Yaskawa INFORM job: OK_R2_O38-47,64(1)(90,180)OKKR.JBI

/JOB
//NAME OK_R2_O38-47,64(1)(90,180)OKKR
///FOLDERNAME X4
//POS
///NPOS 669,669,669,19,0,0
///TOOL 0
///POSTYPE PULSE
///PULSE
C00000=90909,-97924,-91406,33882,56334,-85304
C00001=105552,-103822,-93612,26444,49613,-80458
C00002=93803,-39674,-61862,-10952,72624,-83592
C00003=83044,29645,-6844,-3671,113202,-83073
C00004=80232,46018,13481,-1640,119259,-82796
C00005=84341,50404,17488,7249,115666,-79799
C00006=84629,52012,20689,7225,114506,-79766
C00007=84629,51890,21633,7182,113865,-79809
C00008=84629,52012,20689,7225,114506,-79766
C00009=84940,55701,25098,7229,113667,-79705
C00010=84940,55628,25812,7200,113194,-79735
C00011=84829,53963,24073,7195,113413,-79762
C00012=84779,55348,25092,7189,113502,-79775
C00013=83953,58737,25467,6224,116924,-79977
C00014=90636,-6579,-39383,-4621,91502,-82162
C00015=107016,-16132,-49825,-8384,94240,-77109
C00016=106659,-18282,-50653,15937,87636,-73637
C00017=135463,84611,26036,8427,98138,-63561
C00018=135459,73950,19227,14779,115232,-60625
C00019=121103,67404,21507,14676,120976,-65247
C00020=121102,66967,23101,14477,119807,-65411
C00021=121102,66637,23738,14388,119264,-65486
C00022=121102,66967,23101,14477,119807,-65411
C00023=120221,69773,26406,14234,119379,-65811
C00024=120221,69412,27152,14135,118755,-65896
C00025=120511,68181,25704,14224,118959,-65756
C00026=120221,69412,27152,14135,118755,-65896
C00027=120195,60975,7913,14673,121769,-65482
C00028=135454,84776,26243,8428,98096,-63567
C00029=106659,-18282,-50653,15937,87636,-73637
C00030=89310,-122172,-106686,13361,50676,-45199
C00031=123165,-113898,-119110,-19125,43336,19368
C00032=123668,-102412,-109547,-19577,43467,19587
C00033=131184,63359,57441,-15233,67840,18691
C00034=122068,78147,74274,-12505,69533,15106
C00035=122051,87849,89370,-12875,65325,15559
C00036=122051,89227,92048,-12969,64408,15664
C00037=122316,85057,86118,-12868,65923,15592
C00038=122667,82911,83414,-12880,66527,15655
C00039=122667,83831,85320,-12946,65844,15732
C00040=122426,86931,89254,-12983,65000,15737
C00041=122963,79390,78884,-12845,67528,15654
C00042=130632,64185,60223,-15235,66493,18662
C00043=131662,58983,54996,-15425,67212,18954
C00044=131668,55339,42428,-14901,72880,18222
C00045=146861,-92393,-105699,-36485,53490,27620
C00046=148000,-101656,-114811,-36865,54640,27702
C00047=148000,-101656,-114811,-36865,54640,27702
C00048=148000,-101656,-114811,-36865,54640,27702
C00049=159496,-161049,-136264,-30615,73499,21221
C00050=103228,-122632,-133352,7038,92284,523
C00051=103228,-122632,-133352,7038,92284,523
C00052=103228,-124480,-131601,7026,90271,411
C00053=103391,-121920,-131082,6996,91247,517
C00054=103853,-115329,-128981,6922,93290,780
C00055=103391,-120798,-132087,7006,92433,583
C00056=104641,-114737,-130152,6774,94243,1084
C00057=104641,-114737,-130152,6774,94243,1084
C00058=104641,-116137,-129119,6762,92896,1012
C00059=104641,-115940,-129279,6764,93095,1023
C00060=105111,-108950,-126961,6694,95208,1287
C00061=104576,-115792,-130426,6785,93876,1044
C00062=103741,-127928,-135528,6927,90867,609
C00063=103741,-127928,-135528,6927,90867,609
C00064=103741,-127928,-135528,6927,90867,609
C00065=103865,-116944,-129962,6921,93061,771
C00066=103865,-118485,-128547,6909,91408,679
C00067=103865,-118011,-129031,6913,91946,709
C00068=104350,-111197,-126797,6823,94018,978
C00069=103645,-119716,-131347,6963,92509,670
C00070=126331,-111187,-127566,2170,93341,7936
C00071=126314,-110675,-127191,2173,93374,7931
C00072=126314,-111741,-126360,2171,92316,7913
C00073=126314,-111248,-126762,2172,92816,7922
C00074=126152,-104604,-124481,2216,94828,7909
C00075=126314,-111061,-126906,2173,93001,7925
C00076=125902,-111149,-126935,2263,92984,7794
C00077=132196,-109284,-126305,-2386,93568,14490
C00078=132014,-110397,-125220,-2342,92324,14457
C00079=132014,-111538,-124094,-2340,91046,14481
C00080=132014,-110972,-124684,-2340,91699,14468
C00081=131346,-109003,-124013,-2196,92280,14246
C00082=132122,-112463,-125993,-2364,91740,14502
C00083=130696,-128652,-136015,-2037,89553,14081
C00084=130696,-128652,-136015,-2037,89553,14081
C00085=134573,-129962,-127961,-2886,84044,15460
C00086=135247,-123905,-124729,-3029,85191,15657
C00087=135247,-124242,-122895,-3032,83891,15687
C00088=135059,-121526,-122583,-2986,85086,15595
C00089=134621,-115318,-120572,-2888,87018,15405
C00090=135273,-124345,-124575,-3033,84868,15671
C00091=101634,-140552,-130463,4330,80438,4385
C00092=100831,-135445,-127742,4507,81431,4148
C00093=100831,-135220,-126147,4516,80567,4118
C00094=100831,-135304,-126661,4513,80840,4129
C00095=101541,-127818,-124438,4340,83274,4455
C00096=100689,-136992,-128168,4541,80909,4084
C00097=101700,-117063,-135109,4321,95328,4920
C00098=101700,-117063,-135109,4321,95328,4920
C00099=107464,-106510,-121453,3057,92107,6652
C00100=105693,-105772,-119256,3437,91202,6062
C00101=105693,-106748,-117862,3435,89847,6024
C00102=105693,-106325,-118509,3436,90460,6041
C00103=104724,-99451,-116018,3652,92493,5788
C00104=105563,-106984,-120499,3466,91350,6023
C00105=97637,-124436,-133710,5150,90918,3458
C00106=101700,-117063,-135109,4321,95328,4920
C00107=101700,-117063,-135109,4321,95328,4920
C00108=113885,-115939,-123860,1658,88568,8649
C00109=113885,-115976,-123799,1658,88510,8649
C00110=113885,-116503,-122835,1658,87648,8639
C00111=113928,-115223,-122529,1647,88114,8658
C00112=114061,-111130,-121156,1620,89368,8717
C00113=113613,-117192,-124203,1715,88138,8556
C00114=77135,-109099,-124316,9289,94737,-2930
C00115=77964,-100968,-118468,9143,95217,-2626
C00116=77964,-101677,-117713,9127,94398,-2685
C00117=77964,-101560,-117850,9129,94540,-2675
C00118=78928,-97543,-116360,8967,95572,-2290
C00119=77908,-100245,-119438,9173,96179,-2574
C00120=71973,-123086,-130703,10190,92110,-4818
C00121=61369,-106979,-129386,-18745,110548,43775
C00122=54050,-118433,-122678,-29834,105379,66043
C00123=54050,-118432,-122677,-29849,105379,66042
C00124=52380,-128849,-120518,-29019,98947,67079
C00125=52380,-128559,-118965,-28945,98241,67262
C00126=52380,-128751,-119946,-28990,98681,67146
C00127=50245,-132811,-121152,-28917,96763,66805
C00128=52380,-128751,-119946,-28990,98681,67146
C00129=49374,-119498,-117890,-29381,100712,65454
C00130=49135,-119946,-117683,-29342,100317,65463
C00131=49135,-119959,-116418,-29258,99629,65643
C00132=49135,-119963,-116925,-29289,99902,65571
C00133=47420,-122909,-117861,-29192,98489,65269
C00134=49767,-118756,-118042,-29437,101266,65461
C00135=58824,-127197,-127906,-29549,105900,67783
C00136=58824,-127197,-127906,-29549,105900,67783
C00137=55789,-138532,-125635,-28743,98511,68512
C00138=54845,-137144,-123724,-28738,97781,68329
C00139=54845,-136558,-122036,-28679,97131,68490
C00140=54845,-136878,-122937,-28709,97474,68406
C00141=52687,-141381,-124200,-28678,95380,68093
C00142=56052,-135036,-125386,-28893,100051,68223
C00143=56052,-135036,-125386,-28893,100051,68223
C00144=54923,-136926,-123517,-28734,97796,68355
C00145=54923,-136449,-122129,-28684,97260,68488
C00146=54923,-136715,-122887,-28711,97551,68416
C00147=52628,-141500,-124230,-28677,95326,68085
C00148=54923,-138669,-131970,-29176,101590,67387
C00149=49576,-128334,-132403,-27234,106270,69223
C00150=44922,-139442,-128392,-26353,97465,69516
C00151=43106,-142181,-127565,-26251,95168,69348
C00152=43106,-141292,-125343,-26201,94348,69532
C00153=43106,-141708,-126356,-26223,94717,69449
C00154=42222,-150085,-128620,-26118,91814,69764
C00155=43106,-141708,-126356,-26223,94717,69449
C00156=58006,-149727,-131155,-24086,101568,78058
C00157=67130,-160484,-130477,-19696,102779,86761
C00158=65530,-164092,-131264,-20694,100171,85228
C00159=25938,-108868,-115377,-27148,106727,70167
C00160=30236,-167786,-131335,-27861,77157,62843
C00161=40913,-181249,-136978,-30366,76641,63974
C00162=31337,-124593,-132531,-25311,107075,53461
C00163=107165,-96970,-126665,3187,100215,6761
C00164=107165,-106401,-121090,3121,91950,6553
C00165=98999,-123975,-120325,10477,76714,-326
C00166=104449,-120152,-119012,8815,77213,1590
C00167=136338,-77147,-102883,-1281,87901,12266
C00168=129257,-75496,-102169,6212,88982,4910
C00169=138081,-104464,-122106,-1833,85725,12838
C00170=119260,-105046,-123410,8534,87528,2432
C00171=124620,-151805,-134891,7305,72242,3267
C00172=124614,-151414,-134787,7302,72378,3273
C00173=124612,-151215,-134734,7300,72449,3276
C00174=124620,-151805,-134891,7305,72242,3267
C00175=127969,-108981,-129625,6073,90620,5362
C00176=128058,-112032,-130642,6044,89675,5344
C00177=99990,-117497,-120264,13536,83880,-4252
C00178=95862,-116029,-118012,14517,83962,-5647
C00179=139101,-101989,-113180,2891,83526,8647
C00180=134512,-124069,-125019,4259,79673,7022
C00181=124704,-125859,-130096,7035,82535,3892
C00182=99313,-127153,-133045,-12119,95446,32872
C00183=57886,-133831,-130402,-29291,103936,67934
C00184=55789,-138532,-125635,-28743,98511,68512
C00185=48693,-117877,-116324,-29063,104784,69163
C00186=50073,-120833,-117390,-28223,106210,71565
C00187=68626,-163926,-129258,-19114,104295,87122
C00188=70376,-133538,-127464,-20847,118406,85282
C00189=70376,-133538,-127464,-20847,118406,85282
C00190=56915,-96442,-108782,-30239,105442,63415
C00191=56121,-79134,-101591,-31100,116741,68778
C00192=90261,-137084,-122094,-21625,111979,84005
C00193=77475,-118139,-116359,-17026,122373,89952
C00194=79183,-112936,-123408,-17693,125433,82686
C00195=81561,-124200,-134149,-21063,125175,90603
C00196=103376,-109759,-132308,3968,97270,5504
C00197=101634,-140552,-130463,4330,80438,4385
C00198=110110,-127209,-124061,-3201,83105,15977
C00199=90594,-117032,-120596,11082,89723,-6771
C00200=125366,-116446,-120359,4331,86595,4547
C00201=114221,-95322,-113096,13979,98696,-11684
C00202=109678,-119625,-133746,14623,99658,-13079
C00203=112326,-124641,-135293,14185,97639,-12436
C00204=113675,-111285,-124420,14007,97585,-11993
C00205=113699,-111426,-124467,14002,97539,-11990
C00206=124004,-129907,-130136,8507,87303,-2218
C00207=139431,-131601,-130697,-461,84652,11785
C00208=149048,-100082,-120338,-2575,94643,14766
C00209=149098,-100150,-120363,-2585,94625,14781
C00210=144513,-99899,-120272,-1580,94586,13343
C00211=148184,-92878,-117624,-2396,96648,14454
C00212=154718,-145008,-134516,-3815,80522,16974
C00213=155631,-143491,-134098,-4008,81086,17267
C00214=123104,-120086,-121421,6334,85998,1376
C00215=127889,-117088,-120449,5327,86600,2988
C00216=148175,-95724,-112847,963,92122,9694
C00217=137316,-91860,-109869,13618,92576,-296
C00218=127829,-127486,-128792,15513,87749,-4031
C00219=127829,-122446,-134816,15592,93826,-3264
C00220=125285,-108995,-105645,-24533,66859,22374
C00221=121876,-100663,-100590,-22961,66967,21017
C00222=120611,-97454,-98556,-22372,66992,20522
C00223=120728,-95778,-96365,-22498,66572,20652
C00224=120611,-97454,-98556,-22372,66992,20522
C00225=120972,-98646,-98782,-22597,66650,20731
C00226=119814,-94892,-97816,-21908,67582,20099
C00227=120972,-98646,-98782,-22597,66650,20731
C00228=122255,-101873,-100811,-23195,66623,21236
C00229=125713,-110249,-105850,-24792,66512,22621
C00230=125414,-109454,-110952,-25434,70557,21724
C00231=121886,-100912,-105844,-23885,70668,20357
C00232=120575,-97642,-103795,-23303,70688,19860
C00233=120636,-96154,-101667,-23400,70203,19982
C00234=120575,-97642,-103795,-23303,70688,19860
C00235=121028,-97980,-103315,-23548,70382,20093
C00236=119871,-93906,-102218,-22897,71374,19458
C00237=121028,-97980,-103315,-23548,70382,20093
C00238=122351,-101230,-105354,-24132,70373,20595
C00239=125908,-109706,-110431,-25687,70298,21973
C00240=125468,-108852,-114009,-26132,73198,21211
C00241=121864,-100250,-108878,-24604,73277,19846
C00242=120523,-96969,-106822,-24029,73283,19350
C00243=120543,-95651,-104748,-24106,72739,19471
C00244=120523,-96969,-106822,-24029,73283,19350
C00245=121096,-97384,-106424,-24308,73024,19616
C00246=119937,-93066,-105230,-23683,74062,18974
C00247=121096,-97384,-106424,-24308,73024,19616
C00248=122450,-100644,-108468,-24886,73032,20117
C00249=126090,-109173,-113564,-26418,72994,21493
C00250=126107,-105383,-120588,-25792,78658,20214
C00251=115870,-101424,-121533,41206,90180,3452
C00252=115851,-106682,-115012,41260,85065,1433
C00253=119242,-98694,-109765,40357,84214,2540
C00254=120508,-95652,-107669,40003,83867,2939
C00255=120512,-93942,-105232,40036,83383,2757
C00256=120508,-95652,-107669,40003,83867,2939
C00257=119976,-95300,-106376,40178,83625,2624
C00258=123146,-93912,-105979,39274,82602,3565
C00259=119976,-95300,-106376,40178,83625,2624
C00260=118706,-98291,-108457,40527,83992,2228
C00261=115305,-106116,-113657,41413,84900,1133
C00262=117529,-113204,-110114,15038,59483,-16836
C00263=119860,-102582,-104476,13511,61010,-15725
C00264=120710,-98611,-102232,12973,61516,-15338
C00265=120712,-96036,-99318,13028,61058,-15391
C00266=120710,-98611,-102232,12973,61516,-15338
C00267=120133,-97446,-101425,13271,61707,-15536
C00268=121539,-92419,-99938,12330,63118,-14842
C00269=120133,-97446,-101425,13271,61707,-15536
C00270=119274,-101350,-103659,13810,61233,-15923
C00271=116924,-111770,-109266,15331,59803,-17031
C00272=118012,-90030,-113480,10859,76824,-11039
C00273=121151,-43618,-104634,-1145,105190,4571
C00274=120753,-40362,-99446,-1000,103667,4481
C00275=120604,-39041,-97355,-946,103057,4446
C00276=120606,-40163,-95662,-941,101440,4458
C00277=120604,-39041,-97355,-946,103057,4446
C00278=120772,-35445,-95769,-1008,103931,4483
C00279=120462,-29091,-92658,-908,105279,4391
C00280=120772,-35445,-95769,-1008,103931,4483
C00281=120921,-36668,-97839,-1062,104577,4517
C00282=121319,-39651,-102962,-1210,106200,4605
C00283=108629,-121399,-122702,16889,67135,-14241
C00284=115336,-113367,-105488,19088,53546,-18271
C00285=117865,-102996,-100223,17109,54980,-16930
C00286=118786,-99066,-98108,16412,55481,-16461
C00287=118815,-96798,-95161,16518,54853,-16552
C00288=118786,-99066,-98108,16412,55481,-16461
C00289=119112,-97264,-98148,16039,56331,-16193
C00290=118757,-93015,-97035,15990,57843,-16106
C00291=119112,-97264,-98148,16039,56331,-16193
C00292=123316,-98367,-98161,13561,55035,-14648
C00293=126858,-97217,-97820,11275,54872,-13210
C00294=123316,-98367,-98161,13561,55035,-14648
C00295=122519,-102389,-100318,14180,54451,-15058
C00296=120328,-113051,-105701,15959,52759,-16243
C00297=124093,-110707,-95637,-16539,52225,18162
C00298=121727,-101468,-90458,-14864,53273,16967
C00299=120864,-97923,-88367,-14268,53637,16545
C00300=120864,-95769,-85768,-14357,53158,16613
C00301=120864,-97923,-88367,-14268,53637,16545
C00302=120753,-94948,-87925,-13988,54838,16331
C00303=119636,-91806,-87160,-13170,55764,15745
C00304=120753,-94948,-87925,-13988,54838,16331
C00305=121593,-98445,-90034,-14553,54501,16732
C00306=123889,-107558,-95262,-16133,53518,17861
C00307=123907,-109460,-104253,-15319,57915,17198
C00308=120718,-89127,-94408,93,103364,-81793
C00309=120702,-88967,-86044,90,98299,-81802
C00310=120714,-92346,-83648,90,95088,-81800
C00311=120719,-93530,-82604,90,93837,-81800
C00312=120721,-91291,-79709,90,93204,-81799
C00313=120719,-93530,-82604,90,93837,-81800
C00314=120503,-94372,-82680,81,93451,-81873
C00315=120503,-97134,-83277,81,92401,-81874
C00316=120503,-94372,-82680,81,93451,-81873
C00317=120501,-93212,-83739,81,94699,-81873
C00318=120496,-89894,-86173,82,97902,-81873
C00319=120512,-90208,-94601,84,102927,-81864
C00320=120739,-87258,-85833,92,99047,-81789
C00321=120752,-90752,-83510,91,95822,-81787
C00322=120758,-91982,-82493,91,94564,-81786
C00323=120759,-89478,-79257,91,93861,-81786
C00324=120758,-91982,-82493,91,94564,-81786
C00325=120462,-95334,-83503,80,93464,-81887
C00326=120461,-97919,-84058,79,92477,-81888
C00327=120462,-95334,-83503,80,93464,-81887
C00328=120460,-94163,-84562,80,94717,-81887
C00329=120456,-90813,-86994,80,97935,-81887
C00330=121033,-93279,-128320,-140,99068,4698
C00331=120997,-110061,-117241,-128,83627,4703
C00332=120579,-101211,-110995,-15,84330,4566
C00333=120424,-97983,-108548,25,84483,4515
C00334=120430,-96385,-106046,24,83763,4517
C00335=120424,-97983,-108548,25,84483,4515
C00336=120936,-92390,-106244,-111,85940,4681
C00337=120538,-86818,-104536,-4,87751,4552
C00338=120936,-92390,-106244,-111,85940,4681
C00339=121096,-95373,-108656,-154,85891,4732
C00340=121527,-103462,-114785,-270,85508,4872
C00341=75677,-91018,-121004,38809,104477,3256
C00342=86494,-89564,-122641,29897,102391,4704
C00343=121241,-108971,-117698,-1136,79653,4828
C00344=120728,-99263,-111358,-963,80734,4651
C00345=120539,-95742,-108880,-900,81016,4587
C00346=120543,-94296,-106552,-902,80326,4593
C00347=120539,-95742,-108880,-900,81016,4587
C00348=120728,-93992,-107595,-961,81127,4647
C00349=120728,-90301,-106424,-959,82303,4638
C00350=120728,-93992,-107595,-961,81127,4647
C00351=121024,-97533,-112143,-1058,82109,4735
C00352=121551,-107098,-118478,-1235,81100,4915
C00353=121569,-100080,-124444,-1231,88376,4850
C00354=117898,-83225,-110918,12916,113641,-67504
C00355=119870,-90654,-110250,12481,109228,-67312
C00356=120686,-93336,-109842,12338,107519,-67211
C00357=120688,-92183,-107571,12276,106730,-67294
C00358=120686,-93336,-109842,12338,107519,-67211
C00359=120163,-91649,-109473,12395,108219,-67318
C00360=121681,-97188,-111137,12239,106219,-67001
C00361=120163,-91649,-109473,12395,108219,-67318
C00362=119359,-88923,-109851,12543,109932,-67413
C00363=117416,-81399,-110449,12994,114344,-67589
C00364=120617,-94125,-108136,-8857,121741,-88541
C00365=120616,-94449,-107526,-8800,121205,-88496
C00366=136098,-107181,-107429,-16269,112846,-84409
C00367=120444,-95183,-107742,-8816,120947,-88541
C00368=119761,-91680,-105499,-9024,121288,74873
C00369=120616,-95784,-105179,19399,105655,-65758
C00370=120617,-94769,-108163,19676,107886,-65380
C00371=121686,-93853,-106574,24019,104588,-57765
C00372=120617,-92780,-110041,24421,107344,-57569
C00373=120617,-90665,-112384,24828,109654,-57058
C00374=120619,-82046,-117525,26421,116533,-55408
C00375=120645,-81988,-112872,3577,88664,-15070
C00376=120614,-96077,-90479,-12976,48732,14983
C00377=120612,-93911,-81283,-13967,44304,15634
C00378=120612,-93390,-79613,-14157,43566,15753
C00379=121252,-93346,-79166,-14714,43437,16096
C00380=121500,-95247,-79374,-15137,42660,16355
C00381=120782,-94947,-80724,-14317,43483,15851
C00382=120611,-93982,-79716,-14233,43318,15795
C00383=120612,-95725,-83890,-13821,44941,15536
C00384=121326,-94847,-83951,-14224,45559,15784
C00385=120613,-94980,-84633,-13612,45776,15407
C00386=120613,-95388,-86250,-13438,46540,15293
C00387=120616,-96933,-104006,5046,49827,739
C00388=120616,-97132,-103061,5097,49146,704
C00389=120617,-95323,-101728,5088,49256,711
C00390=120871,-100699,-104338,4972,48087,759
C00391=120795,-98262,-101888,5054,47837,712
C00392=120618,-95198,-103493,5003,50401,770
C00393=121122,-95129,-103646,4600,50501,986
C00394=120617,-97030,-104927,5009,50342,766
C00395=120617,-96757,-105844,4959,51045,801
C00396=120618,-92718,-112658,4589,57292,1090
C00397=108098,-105677,-132023,7461,89264,-328
C00398=80455,-75739,-120669,16714,100968,-7375
C00399=97258,-84752,-105297,10869,90674,-3530
C00400=97358,-86422,-102930,10833,88387,-3696
C00401=97424,-86715,-102018,10818,87679,-3736
C00402=97216,-90521,-102980,10875,86365,-3919
C00403=97404,-84940,-102216,10822,88698,-3655
C00404=120617,-94266,-106774,4665,84598,3614
C00405=111454,-84543,-103018,13521,90962,-7073
C00406=109783,-86139,-104921,12729,90791,-5985
C00407=106092,-100123,-116923,13597,91547,-7106
C00408=102052,-116072,-128299,14497,91044,-8487
C00409=91007,-121504,-125767,15485,91359,-21712
C00410=120613,-95050,-86060,3557,95049,-80550
C00411=120612,-93945,-81838,3544,93023,-80607
C00412=121155,-91942,-79314,3616,92478,-80448
C00413=120652,-94806,-81837,3543,92579,-80606
C00414=120610,-90975,-79567,3544,93151,-80605
C00415=150255,-82598,-75582,4413,93505,-70504
C00416=122384,-91795,-77981,11848,92227,-69969
C00417=120612,-93489,-79991,12120,92904,-70125
C00418=120613,-94640,-84016,12161,94749,-69944
C00419=120614,-96377,-93023,12320,99298,-69491
C00420=120644,-125570,-121052,-6784,67869,-5403
C00421=120615,-96622,-98748,-12572,58745,14095
C00422=120615,-96643,-96984,-12717,57674,14222
C00423=127606,-89142,-93330,-20657,62312,19456
C00424=120926,-99715,-97034,-13118,56212,14526
C00425=120613,-97817,-97899,-12721,57634,14225
C00426=120615,-96818,-95655,6616,54391,866
C00427=120615,-97044,-96976,6561,55085,910
C00428=112093,-90513,-93108,22044,58833,-17349
C00429=120615,-96644,-96112,9528,53512,-9485
C00430=120615,-96653,-97679,9416,54459,-9397
C00431=120616,-95373,-105489,8868,59856,-8934
C00432=117333,-91440,-108817,14098,83709,-30265
C00433=112347,-94381,-87846,22750,99580,-64599
C00434=112329,-92021,-78548,22454,95406,-65402
C00435=115628,-91274,-75119,22621,92902,-64661
C00436=117255,-90241,-73175,22718,91835,-64269
C00437=117028,-88603,-73220,22719,92705,-64185
C00438=116923,-92272,-75451,22697,92259,-64308
C00439=120553,-90828,-77383,-15099,94128,-70510
C00440=120613,-90885,-77384,-15804,94030,-70628
C00441=123770,-105111,-82751,-16580,84167,-79857
C00442=124886,-104010,-85216,-16560,86394,-79763
C00443=120613,-94284,-84162,-15892,96365,-70931
C00444=120614,-95920,-93129,-16139,100869,-71526
C00445=120649,-92160,-111225,-3199,84919,-49711
C00446=120616,-97604,-99172,11891,40402,-23254
C00447=120614,-96911,-90603,13253,35598,-24030
C00448=120614,-96763,-89737,13401,35153,-24111
C00449=121291,-96342,-89250,12683,34963,-23744
C00450=119113,-97762,-90324,15090,35268,-24978
C00451=120705,-99580,-90146,13704,33974,-24279
C00452=121588,-95238,-86691,12692,33949,-23762
C00453=127502,-77730,-88040,-1756,56127,-19882
C00454=125086,-93679,-98074,-150,54079,-20822
C00455=120613,-95818,-85653,14108,33181,-24494
C00456=120615,-97479,-97669,6545,55280,923
C00457=121580,-96410,-96097,5967,54791,1285
C00458=120928,-100587,-97757,6468,53722,953
C00459=120613,-98670,-98620,6548,55254,920
C00460=120615,-96854,-96360,6584,54805,893
C00461=120615,-97074,-97513,6537,55399,931
C00462=114077,-92170,-94328,19163,57465,-15491
C00463=120615,-97626,-97578,9481,53904,-9448
C00464=120636,-112691,-117418,8831,59265,-10492
C00465=120617,-94408,-109491,7961,65698,-13071
C00466=120616,-97035,-102174,8375,59902,-13490
C00467=120616,-97254,-100452,8474,58742,-13580
C00468=120616,-96110,-99125,8495,58514,-13598
C00469=120614,-98453,-101360,8481,58685,-13585
C00470=119727,-100186,-100479,9138,57364,-14041
C00471=120617,-96158,-99373,8483,58642,-13587
C00472=120616,-97215,-100721,8458,58926,-13566
C00473=120616,-96978,-102436,8360,60091,-13476
C00474=120617,-94247,-109716,7948,65917,-13056
C00475=120616,-96445,-103082,-5252,59171,13430
C00476=120615,-96888,-94956,-5569,53965,13694
C00477=120614,-96711,-93127,-5642,52935,13750
C00478=120614,-96618,-92386,-5672,52529,13773
C00479=119756,-94067,-91753,-5051,53390,13370
C00480=120525,-97964,-94062,-5589,52861,13717
C00481=120614,-96681,-92800,-5656,52750,13760
C00482=120614,-96709,-92988,-5648,52851,13755
C00483=120614,-96767,-93400,-5632,53074,13742
C00484=120614,-96843,-94134,-5603,53484,13720
C00485=120615,-96977,-95945,-5531,54526,13664
C00486=120616,-97003,-101109,-6851,58481,13557
C00487=120615,-97139,-99377,-6934,57353,13629
C00488=120615,-97164,-98672,-6968,56909,13657
C00489=119756,-94335,-97933,-6375,57832,13263
C00490=120570,-98373,-100300,-6912,57283,13615
C00491=120615,-97165,-99156,-6946,57204,13638
C00492=120616,-97129,-99856,-6912,57651,13610
C00493=120616,-96964,-101578,-6829,58787,13537
C00494=120617,-96349,-105255,-7716,61917,13386
C00495=120616,-96771,-103611,-7804,60699,13471
C00496=120616,-96905,-102940,-7840,60222,13505
C00497=119756,-93851,-102113,-7266,61195,13116
C00498=120602,-97980,-104523,-7800,60639,13470
C00499=120616,-96844,-103353,-7819,60505,13485
C00500=120616,-96699,-104019,-7783,60985,13451
C00501=120617,-96245,-105652,-7696,62212,13366
C00502=120618,-92150,-112439,-7334,68442,12961
C00503=130920,-122289,-127601,23263,76296,-33617
C00504=126647,-121486,-124764,14921,71090,-19914
C00505=118673,-117816,-113052,9081,54805,-1270
C00506=119719,-97166,-102733,8035,58912,-525
C00507=118944,-92090,-109805,27006,83902,-36269
C00508=120616,-93914,-111601,26462,83549,-35758
C00509=120617,-94475,-108119,24525,75199,-30020
C00510=120618,-90011,-113520,23738,94905,-43572
C00511=120617,-93534,-109718,22404,79768,-31867
C00512=120617,-93028,-110386,24696,84592,-28860
C00513=120617,-93859,-109223,24523,82429,-27907
C00514=120617,-95217,-106728,22357,73913,-21133
C00515=120616,-96198,-104144,16550,64688,-11231
C00516=120616,-97587,-102867,7505,58697,-196
C00517=120615,-98378,-102979,-677,57412,8649
C00518=120615,-98092,-104435,-2505,58558,10610
C00519=120615,-97859,-104607,-2041,58746,10113
C00520=120615,-97689,-104685,-1580,58853,9618
C00521=120615,-97267,-104663,2078,59079,5700
C00522=122185,-96113,-104438,1107,59504,6297
C00523=124417,-94235,-103728,-259,60020,7133
C00524=120617,-96195,-105273,2057,60007,5718
C00525=120617,-95777,-106468,2039,60956,5736
C00526=120690,-30346,-78642,-22937,64170,21118
C00527=120690,-30346,-78642,-22937,64170,21118
C00528=98469,-5770,-79404,-6171,73775,13621
C00529=73961,-64832,-115099,11040,66386,6438
C00530=152983,-151482,-105999,-63266,53723,-19798
C00531=133395,-32083,-56059,-41211,61963,-37621
C00532=138234,23065,45169,-67508,45202,-44915
C00533=136781,30072,55747,-70235,43147,-43411
C00534=136213,33214,60449,-71542,42329,-42699
C00535=136213,31591,57334,-70422,42710,-43384
C00536=136788,30891,57778,-71075,42855,-42892
C00537=134893,29619,56778,-71118,41623,-43172
C00538=133284,25640,52793,-70642,40733,-43707
C00539=131869,22445,49655,-70246,39929,-44150
C00540=132436,19576,45433,-69035,40713,-44782
C00541=133889,13007,35719,-66469,42691,-46136
C00542=120930,8852,32410,-71146,24358,-44597
C00543=120056,16713,42856,-76185,23038,-42237
C00544=121640,23151,50001,-78915,23835,-40720
C00545=120179,17981,45384,-78314,22894,-41190
C00546=119718,18730,44666,-76295,22791,-42223
C00547=126194,31546,58401,-80948,26724,-39140
C00548=125034,24898,50699,-78244,26224,-40637
C00549=126001,16678,39521,-73266,27604,-43020
C00550=110893,28996,24386,-6920,61269,-70362
C00551=121937,-147756,-98721,-13314,47766,-64479
C00552=71720,-152863,-104081,12596,70757,-83485
C00553=71720,-152863,-104081,12596,70757,-83485
C00554=91982,-28216,-51992,-2303,92813,-79298
C00555=103376,51680,-13547,-11468,103274,-76678
C00556=78528,58148,26133,-1884,110066,-82404
C00557=73446,48868,27968,6188,106692,-82975
C00558=73676,48050,29892,6162,105078,-82976
C00559=73848,53549,43602,3176,111557,-82441
C00560=73910,56793,48494,3163,110214,-82456
C00561=74442,47740,29556,6278,105066,-82704
C00562=74442,47438,26373,6344,106859,-82610
C00563=75619,47557,26500,6517,106749,-82195
C00564=75166,47792,29439,6389,105108,-82446
C00565=75942,47613,29246,6502,105072,-82172
C00566=75379,35078,11730,9910,104528,-82166
C00567=80787,8835,-12135,-75,87858,-197
C00568=78204,48375,24964,11405,32429,78205
C00569=74266,-35048,-47468,15580,34736,76255
C00570=76186,-37462,-43585,14686,30875,76605
C00571=72421,-24340,-29465,20568,29825,73730
C00572=72122,-21014,-25782,21301,29384,73365
C00573=70865,-21091,-26712,22563,30208,72759
C00574=70738,-23036,-26859,23341,29404,72363
C00575=73032,-21271,-25966,20119,29138,73940
C00576=72310,-21659,-27383,20648,29949,73692
C00577=73400,-22218,-27785,19257,29646,74366
C00578=78913,-22240,-26725,-522,27359,85032
C00579=79845,-22599,-26982,-1923,27347,85705
C00580=74626,-21952,-29259,17095,30372,75430
C00581=71216,-28758,-34962,21414,31172,73342
C00582=77326,-37520,-49068,12046,33946,77926
C00583=83330,-46575,-52890,13958,55049,41505
C00584=86193,-52033,-54165,20785,79907,-1804
C00585=87571,-35325,-52921,25788,81678,-348
C00586=87508,-34952,-39783,27132,74543,-196
C00587=104644,32154,27534,-4448,60513,-72731
C00588=93805,201,18674,-23355,11914,-69008
C00589=93808,216,18686,-23365,11915,-69004
C00590=93810,222,18691,-23369,11915,-69002
C00591=93638,2355,20486,-22861,11860,-69245
C00592=93955,-2017,16089,-22978,12371,-69170
C00593=93808,210,18682,-23363,11914,-69005
C00594=93806,198,18671,-23357,11914,-69008
C00595=93804,186,18662,-23351,11913,-69011
C00596=93802,180,18657,-23347,11913,-69012
C00597=93799,166,18644,-23338,11912,-69017
C00598=93810,232,18700,-23265,11906,-69051
C00599=95314,-4751,13530,-26418,12915,-67513
C00600=95472,472,19818,-29385,11915,-66147
C00601=93990,-1863,16961,-23823,11950,-68785
C00602=93814,-607,16661,-21825,12670,-69707
C00603=101206,3306,22214,-43193,14297,-59419
C00604=100936,-4761,10472,-35572,16592,-62958
C00605=101724,-18723,-6868,-31140,19848,-65000
C00606=104644,32154,27534,-4448,60513,-72731
C00607=81813,-56841,-53371,53266,50302,-14082
C00608=60380,-131230,-84967,114894,34586,-40161
C00609=75788,-111312,-115723,41491,75595,-63087
C00610=90161,-54224,-109841,-7916,106787,-80704
C00611=104839,2947,-47825,-15873,91805,-74161
C00612=89900,18802,-35938,-9766,95357,-80687
C00613=83481,65005,13429,9056,119285,-78997
C00614=84379,59258,13120,8878,116463,-78905
C00615=105122,63991,30490,-2309,126100,-76457
C00616=105343,61862,26796,-2259,127285,-76391
C00617=86425,59542,13444,9048,116200,-78190
C00618=84859,64061,16437,8959,116837,-78702
C00619=84733,23156,-31643,6898,102580,-79911
C00620=89806,-37631,-52942,-13196,44828,-72538
C00621=94750,-32934,-45091,-18174,44929,-69862
C00622=95076,-26053,-35452,-19245,42727,-69219
C00623=107305,-33153,-35053,-31246,31625,-63156
C00624=107702,-34958,-34985,-32523,30946,-62498
C00625=98239,-24688,-34495,-21885,43616,-67814
C00626=95242,-30076,-40811,-18964,43932,-69406
C00627=95187,-81119,-79791,-20309,40550,-69551
C00628=116770,-29253,-58359,-25644,67366,-65351
C00629=114505,57687,20883,1024,117266,-70683
C00630=114650,58283,25572,1570,115664,-70627
C00631=114340,74668,47492,6514,119432,-70541
C00632=114056,77377,51999,6323,118081,-70732
C00633=114904,58629,25963,1620,115597,-70533
C00634=114904,58844,24763,1634,116445,-70521
C00635=115700,60684,26853,1789,116088,-70230
C00636=115527,59563,26959,1744,115454,-70303
C00637=116183,60608,28143,1870,115246,-70063
C00638=116183,61347,24564,1918,117826,-70018
C00639=115340,32559,-12600,852,114283,-70930
C00640=136323,52272,9545,-44589,64919,-61463
C00641=135074,-39507,-20212,-67575,45484,-47636
C00642=135318,-36807,-17542,-67853,45540,-47442
C00643=132787,-33499,-8836,-71025,42480,-45664
C00644=136770,-25555,-2359,-71345,45178,-45070
C00645=137559,-27867,-5282,-70853,45921,-45309
C00646=137893,-26315,-4086,-70829,46171,-45290
C00647=138309,-31340,-10754,-69522,47005,-46113
C00648=134147,-41542,-18435,-69427,44030,-46529
C00649=141128,-29133,-31085,-43489,44991,-50173
C00650=141423,-23417,-25276,-46918,44761,-56943
C00651=142721,-20298,-19655,-49027,44184,-55636
C00652=146072,-18893,-14822,-60688,47208,-48761
C00653=145286,-17068,-12207,-60970,46372,-48581
C00654=147042,-10361,-12167,-50830,46887,-54547
C00655=146980,-8744,-14162,-48811,51872,-51880
C00656=141391,-26070,-33699,-44316,51156,-54843
C00657=135350,-43982,-50251,-40364,49000,-57185
C00658=135985,2271,-36804,9338,77862,-64370
C00659=125855,24131,-11164,15237,94532,-65211
C00660=127405,33399,-2104,16711,101562,-63562
C00661=127405,32756,72,16600,99959,-63785
C00662=132541,67844,41901,19973,110951,-60327
C00663=132116,69898,43068,19947,111372,-60417
C00664=131318,40837,8366,16232,98288,-62662
C00665=131725,32981,-1351,15245,94948,-63065
C00666=135145,-3466,-36539,10688,79487,-64114
C00667=125690,-78122,-87562,13631,67908,-68588
C00668=2173,-78122,-87562,13631,67908,-68588
BC00000=277574,497829,168108
BC00001=277574,439333,87994
BC00002=272426,396216,154258
BC00003=276020,397785,163842
BC00004=276959,398195,166346
BC00005=274741,403082,149056
BC00006=274741,403082,149056
BC00007=274741,403082,149056
BC00008=274741,403082,149056
BC00009=274741,403082,149056
BC00010=274741,403082,149056
BC00011=274741,403082,149056
BC00012=274741,403082,149056
BC00013=275374,402065,146063
BC00014=277200,399025,164359
BC00015=277200,399025,164359
BC00016=277574,398402,168108
BC00017=337058,429692,17
BC00018=337058,399419,13781
BC00019=288570,380415,46933
BC00020=288570,380415,46933
BC00021=288570,380415,46933
BC00022=288570,380415,46933
BC00023=288570,380415,46933
BC00024=288570,380415,46933
BC00025=288570,380415,46933
BC00026=288570,380415,46933
BC00027=288570,380415,46933
BC00028=326292,423556,17
BC00029=277574,398402,168108
BC00030=248570,470524,121847
BC00031=96843,506307,308542
BC00032=96843,434340,293706
BC00033=128699,374993,308542
BC00034=128699,360593,308542
BC00035=128699,360593,308542
BC00036=128699,360593,308542
BC00037=128699,360593,308542
BC00038=128699,360593,308542
BC00039=128699,360593,308542
BC00040=128699,360593,308542
BC00041=128699,360593,308542
BC00042=128699,370385,308542
BC00043=128699,370385,308542
BC00044=128699,370385,308542
BC00045=128699,434340,293706
BC00046=128699,506307,308542
BC00047=128699,506307,1074774
BC00048=128699,506307,1074774
BC00049=10685,307107,1074774
BC00050=2446,176929,1073423
BC00051=90,176033,1058429
BC00052=90,176033,1058429
BC00053=90,176033,1058429
BC00054=90,176033,1058429
BC00055=90,176033,1058429
BC00056=75724,192083,1061957
BC00057=76484,191603,1056714
BC00058=76484,191603,1056714
BC00059=76484,191603,1056714
BC00060=76484,191603,1056714
BC00061=76484,191603,1056714
BC00062=76484,191603,1056714
BC00063=62310,231239,1056714
BC00064=67554,227591,1021238
BC00065=67554,227591,1021238
BC00066=67554,227591,1021238
BC00067=67554,227591,1021238
BC00068=67554,227591,1021235
BC00069=67554,227591,1021238
BC00070=67554,227591,1021238
BC00071=67554,227591,1021238
BC00072=67554,227591,1021238
BC00073=67554,227591,1021238
BC00074=67554,227591,1021238
BC00075=67554,227591,1021238
BC00076=145464,246213,1073324
BC00077=166805,220817,1072040
BC00078=166805,220817,1072040
BC00079=166805,220817,1072040
BC00080=166805,220817,1072040
BC00081=166805,220817,1072040
BC00082=166805,220817,1072040
BC00083=166804,220816,1072039
BC00084=274112,228208,1072039
BC00085=274112,228208,1072039
BC00086=274112,228208,1072039
BC00087=274112,228208,1072039
BC00088=274112,228208,1072039
BC00089=274112,228208,1072039
BC00090=274112,228208,1072039
BC00091=274112,228208,1072039
BC00092=274112,228208,1072035
BC00093=274112,228208,1072035
BC00094=274112,228208,1072035
BC00095=274112,228208,1072035
BC00096=274112,228208,1072035
BC00097=274112,228208,1072035
BC00098=253771,294542,1072035
BC00099=253771,294542,1066351
BC00100=253771,294542,1066351
BC00101=253771,294542,1066351
BC00102=253771,294542,1066351
BC00103=253771,294542,1066351
BC00104=253771,294542,1066351
BC00105=253771,294542,1066351
BC00106=332674,307450,1072035
BC00107=352760,246268,1062013
BC00108=352760,246268,1056084
BC00109=352760,246268,1056084
BC00110=352760,246268,1056084
BC00111=352760,246268,1056084
BC00112=352760,246268,1056084
BC00113=352760,246268,1056084
BC00114=352760,246268,1056084
BC00115=352760,246268,1056084
BC00116=352760,246268,1056084
BC00117=352760,246268,1056084
BC00118=352760,246268,1056084
BC00119=352760,246268,1056084
BC00120=352760,246268,1056084
BC00121=310153,278141,1073433
BC00122=291607,278327,1074936
BC00123=268886,285111,1073169
BC00124=268886,285111,1073169
BC00125=268886,285111,1073169
BC00126=268886,285111,1073169
BC00127=268886,285111,1073169
BC00128=268886,285111,1073169
BC00129=320862,285111,1073169
BC00130=320862,285111,1073169
BC00131=320862,285111,1073169
BC00132=320862,285111,1073169
BC00133=320862,285111,1073169
BC00134=320862,285111,1073169
BC00135=320862,285111,1073169
BC00136=213321,285111,1073169
BC00137=213321,285111,1068759
BC00138=213321,285111,1068759
BC00139=213321,285111,1068759
BC00140=213321,285111,1068759
BC00141=213321,285111,1068759
BC00142=213321,285111,1068759
BC00143=170741,285111,1068759
BC00144=170741,285111,1068759
BC00145=170741,285111,1068759
BC00146=170741,285111,1068759
BC00147=170741,285111,1068759
BC00148=170741,285111,1068759
BC00149=193205,122603,1068759
BC00150=193205,122603,1068759
BC00151=193205,122603,1068759
BC00152=193205,122603,1068759
BC00153=193205,122603,1068759
BC00154=193205,122603,1068759
BC00155=193205,122603,1068759
BC00156=199695,122603,1068758
BC00157=207772,122603,1068756
BC00158=207772,122603,1068754
BC00159=207772,122603,1068756
BC00160=207772,122603,1068756
BC00161=207772,122603,1068756
BC00162=207772,122603,1073551
BC00163=282390,309614,1068519
BC00164=282390,309614,1066351
BC00165=282388,309615,1066351
BC00166=282388,309615,1066351
BC00167=282388,309615,1066351
BC00168=282388,309615,1066351
BC00169=282388,309615,1066351
BC00170=100662,216693,1072303
BC00171=113337,188658,1072303
BC00172=107541,187687,1072404
BC00173=36523,175786,1073647
BC00174=30619,174782,1073647
BC00175=112223,231348,1072404
BC00176=388754,325280,1072404
BC00177=395558,265794,1072402
BC00178=396585,256820,1072402
BC00179=396585,256820,1072402
BC00180=396585,256820,1072402
BC00181=396585,256820,1072402
BC00182=316583,269170,1070812
BC00183=213321,285111,1068759
BC00184=213321,285111,1068759
BC00185=213321,285111,1068759
BC00186=213321,285111,1068759
BC00187=213321,285111,1068759
BC00188=213321,285111,1068759
BC00189=327369,285111,1068759
BC00190=316865,305805,1068759
BC00191=316865,305805,1068759
BC00192=316865,305805,1068759
BC00193=316865,305805,1068759
BC00194=316858,305779,1068759
BC00195=316082,302674,1068759
BC00196=274112,236301,1072039
BC00197=274112,228208,1072039
BC00198=274113,228208,1072037
BC00199=274113,228208,1072037
BC00200=274113,228208,1072037
BC00201=274113,228208,1072037
BC00202=274113,228208,1072037
BC00203=191168,215841,1072037
BC00204=191168,215841,1072037
BC00205=191168,215841,1072037
BC00206=191168,215841,1072037
BC00207=191168,215841,1072037
BC00208=191168,215841,1072037
BC00209=191168,215841,1072037
BC00210=181197,215841,1072037
BC00211=181197,215841,1072037
BC00212=181197,215841,1072037
BC00213=102071,227043,1072037
BC00214=102071,227043,1072037
BC00215=102071,227043,1072037
BC00216=102071,227043,1072037
BC00217=102071,227043,1072037
BC00218=102071,227043,1072034
BC00219=124217,449505,1070714
BC00220=168838,345562,1075139
BC00221=168838,345562,1075139
BC00222=168838,345562,1075139
BC00223=168838,345562,1075139
BC00224=168838,345562,1075139
BC00225=168838,345562,1075139
BC00226=168838,345562,1075139
BC00227=168838,345562,1075139
BC00228=168838,345562,1075139
BC00229=168838,345562,1075139
BC00230=125540,323298,1075139
BC00231=125540,323298,1075139
BC00232=125540,323298,1075139
BC00233=125540,323298,1075139
BC00234=125540,323298,1075139
BC00235=125540,323298,1075139
BC00236=125540,323298,1075139
BC00237=125540,323298,1075139
BC00238=125540,323298,1075139
BC00239=125540,323298,1075139
BC00240=94014,306720,1075139
BC00241=94014,306720,1075139
BC00242=94014,306720,1075139
BC00243=94014,306720,1075139
BC00244=94014,306720,1075139
BC00245=94014,306720,1075139
BC00246=94014,306720,1075139
BC00247=94014,306720,1075139
BC00248=94014,306720,1075139
BC00249=94014,306720,1075139
BC00250=94014,306720,1075139
BC00251=254000,289563,1075139
BC00252=254000,289563,1075139
BC00253=254000,289563,1075139
BC00254=254000,289563,1075139
BC00255=254000,289563,1075139
BC00256=254000,289563,1075139
BC00257=254000,289563,1075139
BC00258=254000,289563,1075139
BC00259=254000,289563,1075139
BC00260=254000,289563,1075139
BC00261=254000,289563,1075139
BC00262=131735,327892,1075139
BC00263=131735,327892,1075139
BC00264=131735,327892,1075139
BC00265=131735,327892,1075139
BC00266=131735,327892,1075139
BC00267=131735,327892,1075139
BC00268=131735,327892,1075139
BC00269=131735,327892,1075139
BC00270=131735,327892,1075139
BC00271=131735,327892,1075139
BC00272=107464,322487,1075139
BC00273=36166,306609,1075139
BC00274=36166,306609,1075139
BC00275=36166,306609,1075139
BC00276=36166,306609,1075139
BC00277=36166,306609,1075139
BC00278=36166,306609,1075139
BC00279=36166,306609,1075139
BC00280=36166,306609,1075139
BC00281=36166,306609,1075139
BC00282=36166,306609,1075139
BC00283=65350,327285,1075139
BC00284=79942,337624,1075139
BC00285=79942,337624,1075139
BC00286=79942,337624,1075139
BC00287=79942,337624,1075139
BC00288=79942,337624,1075139
BC00289=79942,337624,1075139
BC00290=79942,337624,1075139
BC00291=79942,337624,1075139
BC00292=79942,337624,1075139
BC00293=79942,337624,1075139
BC00294=79942,337624,1075139
BC00295=79942,337624,1075139
BC00296=79942,337624,1075139
BC00297=253079,394331,1075139
BC00298=253079,394331,1075139
BC00299=253079,394331,1075139
BC00300=253079,394331,1075139
BC00301=253079,394331,1075139
BC00302=253079,394331,1075139
BC00303=253079,394331,1075139
BC00304=253079,394331,1075139
BC00305=253079,394331,1075139
BC00306=253079,394331,1075139
BC00307=253079,394331,1075139
BC00308=277954,417010,1075139
BC00309=277954,417010,1075139
BC00310=277954,417010,1075139
BC00311=277954,417010,1075139
BC00312=277954,417010,1075139
BC00313=277954,417010,1075139
BC00314=277954,417010,1075139
BC00315=277954,417010,1075139
BC00316=277954,417010,1075139
BC00317=277954,417010,1075139
BC00318=277954,417010,1075139
BC00319=277954,417010,1075139
BC00320=391385,416545,1075139
BC00321=391385,416545,1075139
BC00322=391385,416545,1075139
BC00323=391385,416545,1075139
BC00324=391385,416545,1075139
BC00325=391385,416545,1075139
BC00326=391385,416545,1075139
BC00327=391385,416545,1075139
BC00328=391385,416545,1075139
BC00329=391385,416545,1075139
BC00330=391263,327160,1075139
BC00331=391263,327160,1075139
BC00332=391263,327160,1075139
BC00333=391263,327160,1075139
BC00334=391263,327160,1075139
BC00335=391263,327160,1075139
BC00336=391263,327160,1075139
BC00337=391263,327160,1075139
BC00338=391263,327160,1075139
BC00339=391263,327160,1075139
BC00340=391263,327160,1075139
BC00341=356655,324576,1075139
BC00342=337458,323143,1075139
BC00343=275792,318538,1075139
BC00344=275792,318538,1075139
BC00345=275792,318538,1075139
BC00346=275792,318538,1075139
BC00347=275792,318538,1075139
BC00348=275792,318538,1075139
BC00349=275792,318538,1075139
BC00350=275792,318538,1075139
BC00351=275792,318538,1075139
BC00352=275792,318538,1075139
BC00353=275792,318538,1075139
BC00354=307207,279391,1075139
BC00355=307207,279391,1075139
BC00356=307207,279391,1075139
BC00357=307207,279391,1075139
BC00358=307207,279391,1075139
BC00359=307207,279391,1075139
BC00360=307207,279391,1075139
BC00361=307207,279391,1075139
BC00362=307207,279391,1075139
BC00363=307207,279391,1075139
BC00364=285880,255332,1075139
BC00365=287298,259977,1075139
BC00366=287865,261836,1075133
BC00367=287865,261835,1075139
BC00368=287865,261835,1075139
BC00369=331646,281789,1075139
BC00370=298873,264569,1075139
BC00371=304319,267702,1075139
BC00372=306227,266863,1075139
BC00373=310997,264767,1075139
BC00374=310976,264769,1075139
BC00375=288935,352548,1075139
BC00376=272404,418382,1075139
BC00377=272425,418380,1075139
BC00378=274896,411588,1075139
BC00379=275885,408871,1075139
BC00380=275885,408871,1075139
BC00381=275885,408871,1075139
BC00382=271736,406720,1075139
BC00383=238429,389236,1075139
BC00384=234311,387049,1075139
BC00385=233323,389766,1075139
BC00386=230852,396558,1075139
BC00387=77992,329104,1075139
BC00388=77753,321663,1075139
BC00389=77658,318686,1075139
BC00390=77658,318686,1075139
BC00391=77658,318686,1075139
BC00392=23870,310010,1075139
BC00393=19166,309251,1075139
BC00394=19261,312228,1075139
BC00395=19500,319669,1075139
BC00396=19479,319671,1075139
BC00397=326076,334412,1075139
BC00398=326076,334412,1075139
BC00399=398158,337877,1075139
BC00400=398158,332624,1075139
BC00401=398158,330523,1075139
BC00402=398158,330523,1075139
BC00403=398158,330523,1075139
BC00404=371797,320949,1075139
BC00405=367094,320185,1075139
BC00406=367157,322286,1075139
BC00407=367157,322286,1075139
BC00408=367157,322286,1075139
BC00409=360371,333511,1075139
BC00410=311234,414795,1075139
BC00411=310658,418001,1075139
BC00412=310141,419246,1075139
BC00413=310427,419283,1075139
BC00414=310427,419283,1075139
BC00415=310141,419246,1075139
BC00416=281236,418582,1075139
BC00417=281185,417346,1075139
BC00418=283925,414321,1075139
BC00419=283904,414323,1075139
BC00420=277357,365951,1075139
BC00421=275362,351203,1075139
BC00422=277956,344725,1075139
BC00423=279886,343902,1075139
BC00424=278994,342134,1075139
BC00425=278994,342134,1075139
BC00426=308109,346018,1075139
BC00427=270475,339947,1075139
BC00428=273112,340372,1075139
BC00429=273814,343136,1075139
BC00430=275568,350045,1075139
BC00431=275547,350048,1075139
BC00432=324592,376313,1075139
BC00433=398158,415711,1075139
BC00434=398158,415708,1075139
BC00435=398158,418342,1075139
BC00436=398158,418592,1075137
BC00437=398158,419396,1075139
BC00438=398158,419396,1075139
BC00439=345872,416171,1075139
BC00440=391430,416208,1075139
BC00441=395295,416215,1075139
BC00442=395295,416215,1075139
BC00443=395538,411718,1075139
BC00444=395517,411721,1075139
BC00445=244931,389034,1075139
BC00446=66736,362189,1075139
BC00447=66757,362186,1075139
BC00448=63792,355216,1075139
BC00449=62606,352427,1075139
BC00450=62606,352427,1075139
BC00451=62606,352427,1075139
BC00452=65008,351421,1075139
BC00453=67703,350299,1075139
BC00454=67703,350299,1075139
BC00455=71854,360058,1075139
BC00456=97410,343690,1075139
BC00457=97254,340887,1075139
BC00458=97254,340887,1075139
BC00459=97254,340887,1075139
BC00460=92552,340117,1075139
BC00461=61981,335172,1075139
BC00462=64618,335595,1075139
BC00463=65320,338358,1075139
BC00464=84683,338339,1075139
BC00465=124898,338298,1075139
BC00466=124919,338295,1075139
BC00467=122721,331714,1075139
BC00468=121842,329081,1075139
BC00469=121842,329081,1075139
BC00470=121842,329081,1075139
BC00471=124604,327643,1075139
BC00472=125483,330276,1075139
BC00473=127681,336858,1075139
BC00474=127660,336860,1075139
BC00475=204706,375167,1075139
BC00476=204727,375165,1075139
BC00477=206658,368463,1075139
BC00478=207430,365782,1075139
BC00479=207430,365782,1075139
BC00480=207430,365782,1075139
BC00481=204595,364357,1075139
BC00482=203304,363708,1075139
BC00483=200469,362282,1075139
BC00484=199696,364963,1075139
BC00485=197766,371664,1075139
BC00486=159349,352318,1075139
BC00487=161419,345679,1075139
BC00488=162247,343023,1075139
BC00489=162247,343023,1075139
BC00490=162247,343023,1075139
BC00491=158253,340971,1075139
BC00492=157425,343627,1075139
BC00493=155355,350266,1075139
BC00494=121532,332804,1075139
BC00495=123702,326211,1075139
BC00496=124571,323574,1075139
BC00497=124571,323574,1075139
BC00498=124571,323574,1075139
BC00499=120575,321489,1075139
BC00500=119707,324126,1075139
BC00501=117536,330719,1075139
BC00502=117515,330722,1075139
BC00503=246976,293738,1075139
BC00504=220058,312475,1075139
BC00505=181696,339176,1075139
BC00506=181696,339176,1075139
BC00507=238830,289663,1075139
BC00508=238830,289663,1075139
BC00509=233651,302305,1075139
BC00510=233720,275129,1075139
BC00511=230055,300568,1075139
BC00512=233773,293926,1075139
BC00513=229845,301345,1075139
BC00514=221324,316481,1075139
BC00515=203984,331406,1075139
BC00516=181696,339176,1075139
BC00517=163038,339247,1075139
BC00518=145371,331462,1075139
BC00519=143897,330516,1075139
BC00520=142920,329779,1075139
BC00521=147384,329275,1075139
BC00522=147384,329275,1075139
BC00523=147384,329275,1075139
BC00524=147193,332075,1075139
BC00525=146810,337675,1075139
BC00526=162807,451351,1075139
BC00527=162807,451351,1075139
BC00528=162807,451351,1075139
BC00529=162453,521794,1065824
BC00530=132820,467472,395097
BC00531=132820,404412,289502
BC00532=120096,349166,355367
BC00533=120096,349166,355367
BC00534=120096,349166,355367
BC00535=120096,349166,355367
BC00536=120096,349166,355367
BC00537=120096,349166,355367
BC00538=120096,349166,355367
BC00539=120096,349166,355367
BC00540=120096,349166,355367
BC00541=120096,349166,355367
BC00542=112974,349609,322888
BC00543=112974,349609,322888
BC00544=112974,349609,322888
BC00545=112974,349609,322888
BC00546=112974,349609,322888
BC00547=112974,349609,322888
BC00548=112974,349609,322888
BC00549=112974,349609,322888
BC00550=104797,366608,393288
BC00551=104797,366608,393288
BC00552=104797,430028,393288
BC00553=248238,430028,393288
BC00554=216374,478358,217163
BC00555=216368,511187,17
BC00556=245714,422186,174266
BC00557=260513,392935,231537
BC00558=260513,392935,231537
BC00559=268580,376991,262752
BC00560=268580,376991,262752
BC00561=260513,392935,231537
BC00562=260513,392935,231537
BC00563=260513,392935,231537
BC00564=260513,392935,231537
BC00565=260513,392935,231537
BC00566=260513,392935,231537
BC00567=258451,395861,231851
BC00568=192387,503711,140202
BC00569=243242,418762,84715
BC00570=243242,418762,84715
BC00571=243242,418762,84715
BC00572=243241,418762,84712
BC00573=243242,418762,84715
BC00574=243242,418762,84715
BC00575=243241,418762,84712
BC00576=243241,418762,84712
BC00577=243241,418762,84712
BC00578=243241,418762,84712
BC00579=243241,418762,84712
BC00580=243241,418762,84712
BC00581=243242,418762,84715
BC00582=243242,418762,84715
BC00583=216476,467162,225886
BC00584=195258,521784,385204
BC00585=89212,520969,483593
BC00586=85875,420588,393288
BC00587=85875,366608,393288
BC00588=78678,370892,285281
BC00589=80895,365862,266393
BC00590=81782,363851,258838
BC00591=81782,363851,258838
BC00592=81782,363851,258838
BC00593=77651,361535,258871
BC00594=73102,358986,258908
BC00595=68971,356671,258941
BC00596=68084,358683,266495
BC00597=65866,363713,285383
BC00598=89779,352898,285458
BC00599=91994,347868,266570
BC00600=91994,347868,266570
BC00601=92880,345855,259016
BC00602=92880,345855,259016
BC00603=91994,347868,266570
BC00604=92880,345855,259016
BC00605=92880,345855,259016
BC00606=85875,366608,393288
BC00607=85875,425449,393288
BC00608=85875,480683,393288
BC00609=162275,481443,208218
BC00610=248224,482298,17
BC00611=252979,445520,23880
BC00612=263212,426452,33206
BC00613=270120,415783,48504
BC00614=270120,415783,48504
BC00615=289464,385910,91339
BC00616=289464,385910,91339
BC00617=270120,415783,48504
BC00618=270120,415783,48504
BC00619=270403,415347,49130
BC00620=268946,415539,99829
BC00621=269127,415277,97663
BC00622=269127,415277,97663
BC00623=270992,410018,85971
BC00624=270992,410018,85971
BC00625=269127,415277,97663
BC00626=269127,415277,97663
BC00627=268082,415019,99664
BC00628=272839,412136,103361
BC00629=296862,394030,126769
BC00630=297297,393702,127193
BC00631=301241,390729,131036
BC00632=301241,390729,131036
BC00633=297297,393702,127193
BC00634=297297,393702,127193
BC00635=297297,393702,127193
BC00636=297297,393702,127193
BC00637=297297,393702,127193
BC00638=297297,393702,127193
BC00639=301241,390729,131036
BC00640=309438,492154,17820
BC00641=284170,378212,242122
BC00642=284170,378212,242122
BC00643=284170,378212,242122
BC00644=284170,378212,242122
BC00645=284170,378212,242122
BC00646=284170,378212,242122
BC00647=284170,378212,242122
BC00648=284170,378212,242122
BC00649=294949,384072,143351
BC00650=294949,384072,143351
BC00651=294949,384072,143351
BC00652=294949,384072,143351
BC00653=294949,384072,143351
BC00654=294949,384072,143351
BC00655=294949,384072,143351
BC00656=294949,384072,143351
BC00657=294949,384072,143351
BC00658=324711,384461,146976
BC00659=313310,379554,140627
BC00660=322606,377492,137960
BC00661=322606,377492,137960
BC00662=344698,372591,131621
BC00663=344698,372591,131621
BC00664=322606,377492,137960
BC00665=322606,377492,137960
BC00666=322606,377492,137960
BC00667=313075,521651,131618
BC00668=142415,521651,131618
EC00000=-798156,-1296783
EC00001=-798156,-1296783
EC00002=-798156,-1296783
EC00003=-798156,-1296783
EC00004=-798156,-1296783
EC00005=-798156,-1296783
EC00006=-798156,-1296783
EC00007=-798156,-1296783
EC00008=-798156,-1296783
EC00009=-798156,-1296783
EC00010=-798156,-1296783
EC00011=-798156,-1296783
EC00012=-798156,-1296783
EC00013=-798156,-1296783
EC00014=-798156,-1296783
EC00015=-798156,-1296783
EC00016=-798156,-1296783
EC00017=-798156,-1296783
EC00018=-798156,-1296783
EC00019=-798156,-1296783
EC00020=-798156,-1296783
EC00021=-798156,-1296783
EC00022=-798156,-1296783
EC00023=-798156,-1296783
EC00024=-798156,-1296783
EC00025=-798156,-1296783
EC00026=-798156,-1296783
EC00027=-798156,-1296783
EC00028=-798156,-1296783
EC00029=-798156,-1296783
EC00030=-798156,-1296783
EC00031=-798156,-1296783
EC00032=-798156,-1296783
EC00033=-798156,-1296783
EC00034=-798156,-1296783
EC00035=-798156,-1296783
EC00036=-798156,-1296783
EC00037=-798156,-1296783
EC00038=-798156,-1296783
EC00039=-798156,-1296783
EC00040=-798156,-1296783
EC00041=-798156,-1296783
EC00042=-798156,-1296783
EC00043=-798156,-1296783
EC00044=-798156,-1296783
EC00045=-798156,-1296783
EC00046=-798156,-1296783
EC00047=-798156,-1296783
EC00048=-798156,-1296783
EC00049=-798156,-1296783
EC00050=-798155,-1296782
EC00051=-798155,-1296782
EC00052=-798155,-1296782
EC00053=-798155,-1296782
EC00054=-798155,-1296782
EC00055=-798155,-1296782
EC00056=-798155,-1296782
EC00057=-798155,-1296782
EC00058=-798155,-1296782
EC00059=-798155,-1296782
EC00060=-798155,-1296782
EC00061=-798155,-1296782
EC00062=-798155,-1296782
EC00063=-798155,-1296782
EC00064=-798155,-1296782
EC00065=-798155,-1296782
EC00066=-798155,-1296782
EC00067=-798155,-1296782
EC00068=-798154,-1296782
EC00069=-798155,-1296782
EC00070=-798155,-1296782
EC00071=-798155,-1296782
EC00072=-798155,-1296782
EC00073=-798155,-1296782
EC00074=-798155,-1296782
EC00075=-798155,-1296782
EC00076=-798155,-1296782
EC00077=-798155,-1296782
EC00078=-798155,-1296782
EC00079=-798155,-1296782
EC00080=-798155,-1296782
EC00081=-798155,-1296782
EC00082=-798155,-1296782
EC00083=-798154,-1296781
EC00084=-798154,-1296781
EC00085=-798154,-1296781
EC00086=-798154,-1296781
EC00087=-798154,-1296781
EC00088=-798154,-1296781
EC00089=-798154,-1296781
EC00090=-798154,-1296781
EC00091=-798154,-1296781
EC00092=-798153,-1296779
EC00093=-798153,-1296779
EC00094=-798153,-1296779
EC00095=-798153,-1296779
EC00096=-798153,-1296779
EC00097=-798153,-1296779
EC00098=-798153,-1296779
EC00099=-798153,-1296779
EC00100=-798153,-1296779
EC00101=-798153,-1296779
EC00102=-798153,-1296779
EC00103=-798153,-1296779
EC00104=-798153,-1296779
EC00105=-798153,-1296779
EC00106=-798153,-1296779
EC00107=-798153,-1296779
EC00108=-798153,-1296779
EC00109=-798153,-1296779
EC00110=-798153,-1296779
EC00111=-798153,-1296779
EC00112=-798153,-1296779
EC00113=-798153,-1296779
EC00114=-798153,-1296779
EC00115=-798153,-1296779
EC00116=-798153,-1296779
EC00117=-798153,-1296779
EC00118=-798153,-1296779
EC00119=-798153,-1296779
EC00120=-798153,-1296779
EC00121=-798153,-1296779
EC00122=-798153,-1296779
EC00123=-798152,-1296778
EC00124=-798152,-1296778
EC00125=-798152,-1296778
EC00126=-798152,-1296778
EC00127=-798152,-1296778
EC00128=-798152,-1296778
EC00129=-798152,-1296778
EC00130=-798152,-1296778
EC00131=-798152,-1296778
EC00132=-798152,-1296778
EC00133=-798152,-1296778
EC00134=-798152,-1296778
EC00135=-798152,-1296778
EC00136=-798152,-1296778
EC00137=-798152,-1296778
EC00138=-798152,-1296778
EC00139=-798152,-1296778
EC00140=-798152,-1296778
EC00141=-798152,-1296778
EC00142=-798152,-1296778
EC00143=-798152,-1296778
EC00144=-798152,-1296778
EC00145=-798152,-1296778
EC00146=-798152,-1296778
EC00147=-798152,-1296778
EC00148=-798152,-1296778
EC00149=-798152,-1296778
EC00150=-798152,-1296778
EC00151=-798152,-1296778
EC00152=-798152,-1296778
EC00153=-798152,-1296778
EC00154=-798152,-1296778
EC00155=-798152,-1296778
EC00156=-798151,-1296777
EC00157=-798149,-1296776
EC00158=-798148,-1296776
EC00159=-798149,-1296776
EC00160=-798149,-1296776
EC00161=-798149,-1296776
EC00162=-798149,-1296776
EC00163=-798153,-1296779
EC00164=-798153,-1296779
EC00165=-798152,-1296778
EC00166=-798152,-1296778
EC00167=-798152,-1296778
EC00168=-798152,-1296778
EC00169=-798152,-1296778
EC00170=-798152,-1296778
EC00171=-798152,-1296778
EC00172=-798152,-1296778
EC00173=-798152,-1296778
EC00174=-798152,-1296778
EC00175=-798152,-1296778
EC00176=-798152,-1296778
EC00177=-798151,-1296777
EC00178=-798151,-1296777
EC00179=-798151,-1296777
EC00180=-798151,-1296777
EC00181=-798151,-1296777
EC00182=-798151,-1296777
EC00183=-798152,-1296778
EC00184=-798152,-1296778
EC00185=-798152,-1296778
EC00186=-798152,-1296778
EC00187=-798152,-1296778
EC00188=-798152,-1296778
EC00189=-798152,-1296778
EC00190=-798152,-1296778
EC00191=-798152,-1296778
EC00192=-798152,-1296778
EC00193=-798152,-1296778
EC00194=-798152,-1296778
EC00195=-798152,-1296778
EC00196=-798154,-1296781
EC00197=-798154,-1296781
EC00198=-798153,-1296779
EC00199=-798153,-1296779
EC00200=-798153,-1296779
EC00201=-798153,-1296779
EC00202=-798153,-1296779
EC00203=-798153,-1296779
EC00204=-798153,-1296779
EC00205=-798153,-1296779
EC00206=-798153,-1296779
EC00207=-798153,-1296779
EC00208=-798153,-1296779
EC00209=-798153,-1296779
EC00210=-798153,-1296779
EC00211=-798153,-1296779
EC00212=-798153,-1296779
EC00213=-798153,-1296779
EC00214=-798151,-1296778
EC00215=-798153,-1296779
EC00216=-798153,-1296779
EC00217=-798153,-1296779
EC00218=-798152,-1296778
EC00219=-798152,-1296778
EC00220=-975524,-1296783
EC00221=-975524,-1296783
EC00222=-975524,-1296783
EC00223=-975524,-1296783
EC00224=-975524,-1296783
EC00225=-975524,-1296783
EC00226=-975524,-1296783
EC00227=-975524,-1296783
EC00228=-975524,-1296783
EC00229=-975524,-1296783
EC00230=-975524,-1296783
EC00231=-975524,-1296783
EC00232=-975524,-1296783
EC00233=-975524,-1296783
EC00234=-975524,-1296783
EC00235=-975524,-1296783
EC00236=-975524,-1296783
EC00237=-975524,-1296783
EC00238=-975524,-1296783
EC00239=-975524,-1296783
EC00240=-975524,-1296783
EC00241=-975524,-1296783
EC00242=-975524,-1296783
EC00243=-975524,-1296783
EC00244=-975524,-1296783
EC00245=-975524,-1296783
EC00246=-975524,-1296783
EC00247=-975524,-1296783
EC00248=-975524,-1296783
EC00249=-975524,-1296783
EC00250=-975524,-1296783
EC00251=-975524,-1296783
EC00252=-975524,-1296783
EC00253=-975524,-1296783
EC00254=-975524,-1296783
EC00255=-975524,-1296783
EC00256=-975524,-1296783
EC00257=-975524,-1296783
EC00258=-975524,-1296783
EC00259=-975524,-1296783
EC00260=-975524,-1296783
EC00261=-975524,-1296783
EC00262=-975524,-1296783
EC00263=-975524,-1296783
EC00264=-975524,-1296783
EC00265=-975524,-1296783
EC00266=-975524,-1296783
EC00267=-975524,-1296783
EC00268=-975524,-1296783
EC00269=-975524,-1296783
EC00270=-975524,-1296783
EC00271=-975524,-1296783
EC00272=-975524,-1296783
EC00273=-975524,-1296783
EC00274=-975524,-1296783
EC00275=-975524,-1296783
EC00276=-975524,-1296783
EC00277=-975524,-1296783
EC00278=-975524,-1296783
EC00279=-975524,-1296783
EC00280=-975524,-1296783
EC00281=-975524,-1296783
EC00282=-975524,-1296783
EC00283=-975524,-1296783
EC00284=-975524,-1296783
EC00285=-975524,-1296783
EC00286=-975524,-1296783
EC00287=-975524,-1296783
EC00288=-975524,-1296783
EC00289=-975524,-1296783
EC00290=-975524,-1296783
EC00291=-975524,-1296783
EC00292=-975524,-1296783
EC00293=-975524,-1296783
EC00294=-975524,-1296783
EC00295=-975524,-1296783
EC00296=-975524,-1296783
EC00297=-975524,-1296783
EC00298=-975524,-1296783
EC00299=-975524,-1296783
EC00300=-975524,-1296783
EC00301=-975524,-1296783
EC00302=-975524,-1296783
EC00303=-975524,-1296783
EC00304=-975524,-1296783
EC00305=-975524,-1296783
EC00306=-975524,-1296783
EC00307=-975524,-1296783
EC00308=-975524,-1296783
EC00309=-975524,-1296783
EC00310=-975524,-1296783
EC00311=-975524,-1296783
EC00312=-975524,-1296783
EC00313=-975524,-1296783
EC00314=-975524,-1296783
EC00315=-975524,-1296783
EC00316=-975524,-1296783
EC00317=-975524,-1296783
EC00318=-975524,-1296783
EC00319=-975524,-1296783
EC00320=-975524,-1296783
EC00321=-975524,-1296783
EC00322=-975524,-1296783
EC00323=-975524,-1296783
EC00324=-975524,-1296783
EC00325=-975524,-1296783
EC00326=-975524,-1296783
EC00327=-975524,-1296783
EC00328=-975524,-1296783
EC00329=-975524,-1296783
EC00330=-975524,-1296783
EC00331=-975524,-1296783
EC00332=-975524,-1296783
EC00333=-975524,-1296783
EC00334=-975524,-1296783
EC00335=-975524,-1296783
EC00336=-975524,-1296783
EC00337=-975524,-1296783
EC00338=-975524,-1296783
EC00339=-975524,-1296783
EC00340=-975524,-1296783
EC00341=-975524,-1296783
EC00342=-975524,-1296783
EC00343=-975524,-1296783
EC00344=-975524,-1296783
EC00345=-975524,-1296783
EC00346=-975524,-1296783
EC00347=-975524,-1296783
EC00348=-975524,-1296783
EC00349=-975524,-1296783
EC00350=-975524,-1296783
EC00351=-975524,-1296783
EC00352=-975524,-1296783
EC00353=-975524,-1296783
EC00354=-975524,-1296783
EC00355=-975524,-1296783
EC00356=-975524,-1296783
EC00357=-975524,-1296783
EC00358=-975524,-1296783
EC00359=-975524,-1296783
EC00360=-975524,-1296783
EC00361=-975524,-1296783
EC00362=-975524,-1296783
EC00363=-975524,-1296783
EC00364=-975524,-1296783
EC00365=-975524,-1296783
EC00366=-975518,-1296780
EC00367=-975524,-1296783
EC00368=-975524,-1296783
EC00369=-975524,-1296783
EC00370=-975524,-1296783
EC00371=-975524,-1296783
EC00372=-975524,-1296783
EC00373=-975524,-1296783
EC00374=-975524,-1296783
EC00375=-975524,-1296783
EC00376=-975524,-1296783
EC00377=-975524,-1296783
EC00378=-975524,-1296783
EC00379=-975524,-1296783
EC00380=-975524,-1296783
EC00381=-975524,-1296783
EC00382=-975524,-1296783
EC00383=-975524,-1296783
EC00384=-975524,-1296783
EC00385=-975524,-1296783
EC00386=-975524,-1296783
EC00387=-975524,-1296783
EC00388=-975524,-1296783
EC00389=-975524,-1296783
EC00390=-975524,-1296783
EC00391=-975524,-1296783
EC00392=-975524,-1296783
EC00393=-975524,-1296783
EC00394=-975524,-1296783
EC00395=-975524,-1296783
EC00396=-975524,-1296783
EC00397=-975524,-1296783
EC00398=-975524,-1296783
EC00399=-975524,-1296783
EC00400=-975524,-1296783
EC00401=-975524,-1296783
EC00402=-975524,-1296783
EC00403=-975524,-1296783
EC00404=-975524,-1296783
EC00405=-975524,-1296783
EC00406=-975524,-1296783
EC00407=-975524,-1296783
EC00408=-975524,-1296783
EC00409=-975524,-1296783
EC00410=-975524,-1296783
EC00411=-975524,-1296783
EC00412=-975524,-1296783
EC00413=-975524,-1296783
EC00414=-975524,-1296783
EC00415=-975524,-1296783
EC00416=-975524,-1296783
EC00417=-975524,-1296783
EC00418=-975524,-1296783
EC00419=-975524,-1296783
EC00420=-975524,-1296783
EC00421=-975524,-1296783
EC00422=-975524,-1296783
EC00423=-975524,-1296783
EC00424=-975524,-1296783
EC00425=-975524,-1296783
EC00426=-975524,-1296783
EC00427=-975524,-1296783
EC00428=-975524,-1296783
EC00429=-975524,-1296783
EC00430=-975524,-1296783
EC00431=-975524,-1296783
EC00432=-975524,-1296783
EC00433=-975524,-1296783
EC00434=-975524,-1296783
EC00435=-975524,-1296783
EC00436=-975522,-1296782
EC00437=-975524,-1296783
EC00438=-975524,-1296783
EC00439=-975524,-1296783
EC00440=-975524,-1296783
EC00441=-975524,-1296783
EC00442=-975524,-1296783
EC00443=-975524,-1296783
EC00444=-975524,-1296783
EC00445=-975524,-1296783
EC00446=-975524,-1296783
EC00447=-975524,-1296783
EC00448=-975524,-1296783
EC00449=-975524,-1296783
EC00450=-975524,-1296783
EC00451=-975524,-1296783
EC00452=-975524,-1296783
EC00453=-975524,-1296783
EC00454=-975524,-1296783
EC00455=-975524,-1296783
EC00456=-975524,-1296783
EC00457=-975524,-1296783
EC00458=-975524,-1296783
EC00459=-975524,-1296783
EC00460=-975524,-1296783
EC00461=-975524,-1296783
EC00462=-975524,-1296783
EC00463=-975524,-1296783
EC00464=-975524,-1296783
EC00465=-975524,-1296783
EC00466=-975524,-1296783
EC00467=-975524,-1296783
EC00468=-975524,-1296783
EC00469=-975524,-1296783
EC00470=-975524,-1296783
EC00471=-975524,-1296783
EC00472=-975524,-1296783
EC00473=-975524,-1296783
EC00474=-975524,-1296783
EC00475=-975524,-1296783
EC00476=-975524,-1296783
EC00477=-975524,-1296783
EC00478=-975524,-1296783
EC00479=-975524,-1296783
EC00480=-975524,-1296783
EC00481=-975524,-1296783
EC00482=-975524,-1296783
EC00483=-975524,-1296783
EC00484=-975524,-1296783
EC00485=-975524,-1296783
EC00486=-975524,-1296783
EC00487=-975524,-1296783
EC00488=-975524,-1296783
EC00489=-975524,-1296783
EC00490=-975524,-1296783
EC00491=-975524,-1296783
EC00492=-975524,-1296783
EC00493=-975524,-1296783
EC00494=-975524,-1296783
EC00495=-975524,-1296783
EC00496=-975524,-1296783
EC00497=-975524,-1296783
EC00498=-975524,-1296783
EC00499=-975524,-1296783
EC00500=-975524,-1296783
EC00501=-975524,-1296783
EC00502=-975524,-1296783
EC00503=-975524,-1296783
EC00504=-975524,-1296783
EC00505=-975524,-1296783
EC00506=-975524,-1296783
EC00507=-975524,-1296783
EC00508=-975524,-1296783
EC00509=-975524,-1296783
EC00510=-975524,-1296783
EC00511=-975524,-1296783
EC00512=-975524,-1296783
EC00513=-975524,-1296783
EC00514=-975524,-1296783
EC00515=-975524,-1296783
EC00516=-975524,-1296783
EC00517=-975524,-1296783
EC00518=-975524,-1296783
EC00519=-975524,-1296783
EC00520=-975524,-1296783
EC00521=-975524,-1296783
EC00522=-975524,-1296783
EC00523=-975524,-1296783
EC00524=-975524,-1296783
EC00525=-975524,-1296783
EC00526=-975524,-1296783
EC00527=-798156,-1296783
EC00528=-798156,-1296783
EC00529=-798154,-1296783
EC00530=-798156,-1296783
EC00531=-798156,-1296783
EC00532=-798156,-1296783
EC00533=-798156,-1296783
EC00534=-798156,-1296783
EC00535=-798156,-1296783
EC00536=-798156,-1296783
EC00537=-798156,-1296783
EC00538=-798156,-1296783
EC00539=-798156,-1296783
EC00540=-798156,-1296783
EC00541=-798156,-1296783
EC00542=-798156,-1296783
EC00543=-798156,-1296783
EC00544=-798156,-1296783
EC00545=-798156,-1296783
EC00546=-798156,-1296783
EC00547=-798156,-1296783
EC00548=-798156,-1296783
EC00549=-798156,-1296783
EC00550=-798156,-1296783
EC00551=-798156,-1296783
EC00552=-798156,-1296783
EC00553=-798156,-1296783
EC00554=-798156,-1296783
EC00555=-798156,-1296783
EC00556=-798156,-1296783
EC00557=-798156,-1296783
EC00558=-798156,-1296783
EC00559=-798156,-1296783
EC00560=-798156,-1296783
EC00561=-798156,-1296783
EC00562=-798156,-1296783
EC00563=-798156,-1296783
EC00564=-798156,-1296783
EC00565=-798156,-1296783
EC00566=-798156,-1296783
EC00567=-798156,-1296783
EC00568=-798156,-1296783
EC00569=-798156,-1296783
EC00570=-798156,-1296783
EC00571=-798156,-1296783
EC00572=-798155,-1296781
EC00573=-798156,-1296783
EC00574=-798156,-1296783
EC00575=-798155,-1296781
EC00576=-798155,-1296781
EC00577=-798155,-1296781
EC00578=-798155,-1296781
EC00579=-798155,-1296781
EC00580=-798155,-1296781
EC00581=-798156,-1296783
EC00582=-798156,-1296783
EC00583=-798156,-1296783
EC00584=-798156,-1296783
EC00585=-798156,-1296783
EC00586=-798156,-1296783
EC00587=-798156,-1296783
EC00588=-798156,-1296783
EC00589=-798156,-1296783
EC00590=-798156,-1296783
EC00591=-798156,-1296783
EC00592=-798156,-1296783
EC00593=-798156,-1296783
EC00594=-798156,-1296783
EC00595=-798156,-1296783
EC00596=-798156,-1296783
EC00597=-798156,-1296783
EC00598=-798156,-1296783
EC00599=-798156,-1296783
EC00600=-798156,-1296783
EC00601=-798156,-1296783
EC00602=-798156,-1296783
EC00603=-798156,-1296783
EC00604=-798156,-1296783
EC00605=-798156,-1296783
EC00606=-798156,-1296783
EC00607=-798156,-1296783
EC00608=-798156,-1296783
EC00609=-798156,-1296783
EC00610=-798156,-1296783
EC00611=-798156,-1296783
EC00612=-798156,-1296783
EC00613=-798155,-1296782
EC00614=-798155,-1296782
EC00615=-798156,-1296783
EC00616=-798156,-1296783
EC00617=-798155,-1296782
EC00618=-798155,-1296782
EC00619=-798155,-1296782
EC00620=-798155,-1296782
EC00621=-798155,-1296782
EC00622=-798155,-1296782
EC00623=-798156,-1296783
EC00624=-798156,-1296783
EC00625=-798155,-1296782
EC00626=-798155,-1296782
EC00627=-798155,-1296782
EC00628=-798155,-1296782
EC00629=-798156,-1296783
EC00630=-798156,-1296783
EC00631=-798156,-1296783
EC00632=-798156,-1296783
EC00633=-798156,-1296783
EC00634=-798156,-1296783
EC00635=-798156,-1296783
EC00636=-798156,-1296783
EC00637=-798156,-1296783
EC00638=-798156,-1296783
EC00639=-798156,-1296783
EC00640=-798156,-1296783
EC00641=-798156,-1296783
EC00642=-798156,-1296783
EC00643=-798156,-1296783
EC00644=-798156,-1296783
EC00645=-798156,-1296783
EC00646=-798156,-1296783
EC00647=-798156,-1296783
EC00648=-798156,-1296783
EC00649=-798156,-1296783
EC00650=-798156,-1296783
EC00651=-798156,-1296783
EC00652=-798156,-1296783
EC00653=-798156,-1296783
EC00654=-798156,-1296783
EC00655=-798156,-1296783
EC00656=-798156,-1296783
EC00657=-798156,-1296783
EC00658=-798156,-1296783
EC00659=-798156,-1296783
EC00660=-798156,-1296783
EC00661=-798156,-1296783
EC00662=-798156,-1296783
EC00663=-798156,-1296783
EC00664=-798156,-1296783
EC00665=-798156,-1296783
EC00666=-798156,-1296783
EC00667=-798155,-1296782
EC00668=-798155,-1296782
///POSTYPE BASE
///RECTAN
///RCONF 0,0,0,0,1,0,0,0,0,0,0,0,0,0,0,0,0,0,0,0,0,0,0,0
P00006=2.006,1.622,-0.565,0.0000,0.0000,0.0000
P00021=0.073,2.058,-0.109,0.0000,0.0000,0.0000
P00022=2.006,1.622,-0.565,0.0000,0.0000,0.0000
///RCONF 0,0,0,0,0,0,0,0,0,0,0,0,0,0,0,0,0,0,0,0,0,0,0,0
P00023=-2.957,-4.083,2.762,0.0000,0.0000,0.0000
P00030=-0.014,-0.768,0.131,0.0000,0.0000,0.0000
P00031=-0.170,0.039,-0.647,0.0000,0.0000,0.0000
P00032=-0.423,0.157,3.222,0.0000,0.0000,0.0000
P00033=0.854,-1.099,3.047,0.0000,0.0000,0.0000
///RCONF 0,0,0,0,1,0,0,0,0,0,0,0,0,0,0,0,0,0,0,0,0,0,0,0
P00034=-8.151,9.743,-4.393,0.0000,0.0000,0.0000
///RCONF 0,0,0,0,0,0,0,0,0,0,0,0,0,0,0,0,0,0,0,0,0,0,0,0
P00035=0.390,-0.027,1.040,0.0000,0.0000,0.0000
P00036=-2.434,0.084,0.197,0.0000,0.0000,0.0000
P00037=-1.075,5.090,-3.949,0.0000,0.0000,0.0000
P00038=0.174,-1.527,-10.860,0.0000,0.0000,0.0000
P00039=-0.109,1.838,-0.266,0.0000,0.0000,0.0000
P00040=2.716,-0.016,3.014,0.0000,0.0000,0.0000
P00041=-0.109,0.014,0.966,0.0000,0.0000,0.0000
P00042=-0.220,0.371,-0.613,0.0000,0.0000,0.0000
P00043=-0.179,-5.890,-3.227,0.0000,0.0000,0.0000
P00044=-8.560,-7.557,-5.232,0.0000,0.0000,0.0000
//INST
///DATE 2024/11/18 21:14
///ATTR SC,RW
///GROUP1 RB1,BS1
///GROUP2 ST1
NOP
'OK_r2_O38-47,64(1)(90,180)
'Down
MOVJ C00000 BC00000 VJ=100.00  +MOVJ EC00000 VJ=100.00
MOVJ C00001 BC00001 VJ=100.00  +MOVJ EC00001 VJ=100.00
MOVJ C00002 BC00002 VJ=100.00  +MOVJ EC00002 VJ=100.00
MOVJ C00003 BC00003 VJ=20.00  +MOVJ EC00003 VJ=20.00
'Path S1883
SFTOF3D
MOVJ C00004 BC00004 VJ=100.00  +MOVJ EC00004 VJ=100.00
MOVL C00005 BC00005 V=500.0  +MOVJ EC00005 VJ=100.00
SMOVL C00006 BC00006 V=100.0  +MOVJ EC00006
SREFP 3 C00007 BC00007  +REFP EC00007
CALL JOB:SEARCH-R1-S13D
SET P021 P006
SFTON3D P021
SMOVL C00008 BC00008 V=100.0  +MOVJ EC00008
SMOVL C00009 BC00009 V=100.0  +MOVJ EC00009
SMOVL C00010 BC00010 V=100.0  +MOVJ EC00010
SREFP 3 C00011 BC00011  +REFP EC00011
CALL JOB:SEARCH-R1-S13D
SET P021 P006
SFTON3D P021
SMOVL C00012 BC00012 V=100.0  +MOVJ EC00012
SFTOF3D
MOVL C00013 BC00013 V=400.0  +MOVJ EC00013 VJ=100.00
MOVJ C00014 BC00014 VJ=100.00  +MOVJ EC00014 VJ=100.00
MOVJ C00015 BC00015 VJ=100.00  +MOVJ EC00015 VJ=100.00
MOVJ C00016 BC00016 VJ=100.00  +MOVJ EC00016 VJ=100.00
MOVJ C00017 BC00017 VJ=100.00  +MOVJ EC00017 VJ=100.00
'Path S1884
SFTOF3D
MOVJ C00018 BC00018 VJ=40.00  +MOVJ EC00018 VJ=100.00
MOVL C00019 BC00019 V=400.0  +MOVJ EC00019 VJ=100.00
SMOVL C00020 BC00020 V=100.0  +MOVJ EC00020
SREFP 3 C00021 BC00021  +REFP EC00021
CALL JOB:SEARCH-R1-S13D
SET P022 P006
SFTON3D P022
SMOVL C00022 BC00022 V=100.0  +MOVJ EC00022
SMOVL C00023 BC00023 V=133.3  +MOVJ EC00023
SMOVL C00024 BC00024 V=100.0  +MOVJ EC00024
SREFP 3 C00025 BC00025  +REFP EC00025
CALL JOB:SEARCH-R1-S13D
SET P022 P006
SFTON3D P022
SMOVL C00026 BC00026 V=100.0  +MOVJ EC00026
MOVL C00027 BC00027 V=1000.0  +MOVJ EC00027 VJ=100.00
MOVJ C00028 BC00028 VJ=100.00  +MOVJ EC00028 VJ=100.00
MOVJ C00029 BC00029 VJ=100.00  +MOVJ EC00029 VJ=100.00
MOVJ C00030 BC00030 VJ=100.00  +MOVJ EC00030 VJ=100.00
MOVJ C00031 BC00031 VJ=100.00  +MOVJ EC00031 VJ=100.00
MOVJ C00032 BC00032 VJ=100.00  +MOVJ EC00032 VJ=100.00
'Path S1885
SFTOF3D
MOVJ C00033 BC00033 VJ=100.00  +MOVJ EC00033 VJ=100.00
MOVL C00034 BC00034 V=166.7  +MOVJ EC00034 VJ=100.00
SMOVL C00035 BC00035 V=100.0  +MOVJ EC00035
SREFP 3 C00036 BC00036  +REFP EC00036
CALL JOB:SEARCH-R1-S13D
SET P023 P006
SFTON3D P023
SMOVL C00037 BC00037 V=100.0  +MOVJ EC00037
SMOVL C00038 BC00038 V=166.7  +MOVJ EC00038
SMOVL C00039 BC00039 V=100.0  +MOVJ EC00039
SREFP 3 C00040 BC00040  +REFP EC00040
CALL JOB:SEARCH-R1-S13D
SET P023 P006
SFTON3D P023
SMOVL C00041 BC00041 V=100.0  +MOVJ EC00041
SFTOF3D
MOVL C00042 BC00042 V=400.0  +MOVJ EC00042 VJ=100.00
MOVL C00043 BC00043 V=1000.0  +MOVJ EC00043 VJ=100.00
MOVL C00044 BC00044 V=1000.0  +MOVJ EC00044 VJ=100.00
MOVJ C00045 BC00045 VJ=100.00  +MOVJ EC00045 VJ=100.00
MOVJ C00046 BC00046 VJ=100.00  +MOVJ EC00046 VJ=100.00
MOVJ C00047 BC00047 VJ=100.00  +MOVJ EC00047 VJ=100.00
'NOWY PROGRAM KRIS
MOVJ C00048 BC00048 VJ=100.00  +MOVJ EC00048 VJ=100.00
MOVJ C00049 BC00049 VJ=100.00  +MOVJ EC00049 VJ=100.00
MOVJ C00050 BC00050 VJ=100.00  +MOVJ EC00050 VJ=100.00
SMOVL C00051 BC00051 V=100.0  +MOVJ EC00051
SREFP 3 C00052 BC00052  +REFP EC00052
CALL JOB:SEARCH-R1-S13D
SET P030 P006
SFTON3D P030
SMOVL C00053 BC00053 V=100.0  +MOVJ EC00053
SREFP 3 C00054 BC00054  +REFP EC00054
CALL JOB:SEARCH-R1-S13D
SET P030 P006
SFTON3D P030
SMOVL C00055 BC00055 V=100.0  +MOVJ EC00055
SFTOF3D
MOVJ C00056 BC00056 VJ=100.00  +MOVJ EC00056 VJ=100.00
SMOVL C00057 BC00057 V=100.0  +MOVJ EC00057
SREFP 3 C00058 BC00058  +REFP EC00058
CALL JOB:SEARCH-R1-S13D
SET P031 P006
SFTON3D P031
SMOVL C00059 BC00059 V=100.0  +MOVJ EC00059
SREFP 3 C00060 BC00060  +REFP EC00060
CALL JOB:SEARCH-R1-S13D
SET P031 P006
SFTON3D P031
SMOVL C00061 BC00061 V=100.0  +MOVJ EC00061
SFTOF3D
MOVJ C00062 BC00062 VJ=100.00  +MOVJ EC00062 VJ=100.00
MOVJ C00063 BC00063 VJ=100.00  +MOVJ EC00063 VJ=100.00
MOVJ C00064 BC00064 VJ=100.00  +MOVJ EC00064 VJ=100.00
SMOVL C00065 BC00065 V=100.0  +MOVJ EC00065
SREFP 3 C00066 BC00066  +REFP EC00066
CALL JOB:SEARCH-R1-S13D
SET P032 P006
SFTON3D P032
SMOVL C00067 BC00067 V=100.0  +MOVJ EC00067
SREFP 3 C00068 BC00068  +REFP EC00068
CALL JOB:SEARCH-R1-S13D
SET P032 P006
SFTON3D P032
SMOVL C00069 BC00069 V=100.0  +MOVJ EC00069
SFTOF3D
MOVJ C00070 BC00070 VJ=100.00  +MOVJ EC00070 VJ=100.00
SMOVL C00071 BC00071 V=100.0  +MOVJ EC00071
SREFP 3 C00072 BC00072  +REFP EC00072
CALL JOB:SEARCH-R1-S13D
SET P033 P006
SFTON3D P033
SMOVL C00073 BC00073 V=100.0  +MOVJ EC00073
SREFP 3 C00074 BC00074  +REFP EC00074
CALL JOB:SEARCH-R1-S13D
SET P033 P006
SFTON3D P033
SMOVL C00075 BC00075 V=100.0  +MOVJ EC00075
SFTOF3D
MOVJ C00076 BC00076 VJ=100.00  +MOVJ EC00076 VJ=100.00
MOVJ C00077 BC00077 VJ=100.00  +MOVJ EC00077 VJ=100.00
SMOVL C00078 BC00078 V=100.0  +MOVJ EC00078
SREFP 3 C00079 BC00079  +REFP EC00079
CALL JOB:SEARCH-R1-S13D
SET P034 P006
SFTON3D P034
SMOVL C00080 BC00080 V=100.0  +MOVJ EC00080
SREFP 3 C00081 BC00081  +REFP EC00081
CALL JOB:SEARCH-R1-S13D
SET P034 P006
SFTON3D P034
SMOVL C00082 BC00082 V=100.0  +MOVJ EC00082
SFTOF3D
MOVJ C00083 BC00083 VJ=100.00  +MOVJ EC00083 VJ=100.00
MOVJ C00084 BC00084 VJ=100.00  +MOVJ EC00084 VJ=100.00
MOVJ C00085 BC00085 VJ=100.00  +MOVJ EC00085 VJ=100.00
SMOVL C00086 BC00086 V=100.0  +MOVJ EC00086
SREFP 3 C00087 BC00087  +REFP EC00087
CALL JOB:SEARCH-R1-S13D
SET P035 P006
SFTON3D P035
SMOVL C00088 BC00088 V=100.0  +MOVJ EC00088
SREFP 3 C00089 BC00089  +REFP EC00089
CALL JOB:SEARCH-R1-S13D
SET P035 P006
SFTON3D P035
SMOVL C00090 BC00090 V=100.0  +MOVJ EC00090
SFTOF3D
MOVJ C00091 BC00091 VJ=100.00  +MOVJ EC00091 VJ=100.00
SMOVL C00092 BC00092 V=100.0  +MOVJ EC00092
SREFP 3 C00093 BC00093  +REFP EC00093
CALL JOB:SEARCH-R1-S13D
SET P036 P006
SFTON3D P036
SMOVL C00094 BC00094 V=100.0  +MOVJ EC00094
SREFP 3 C00095 BC00095  +REFP EC00095
CALL JOB:SEARCH-R1-S13D
SET P036 P006
SFTON3D P036
SMOVL C00096 BC00096 V=100.0  +MOVJ EC00096
SFTOF3D
MOVJ C00097 BC00097 VJ=100.00  +MOVJ EC00097 VJ=100.00
MOVJ C00098 BC00098 VJ=100.00  +MOVJ EC00098 VJ=100.00
MOVJ C00099 BC00099 VJ=100.00  +MOVJ EC00099 VJ=100.00
SMOVL C00100 BC00100 V=100.0  +MOVJ EC00100
SREFP 3 C00101 BC00101  +REFP EC00101
CALL JOB:SEARCH-R1-S13D
SET P044 P006
SFTON3D P044
SMOVL C00102 BC00102 V=100.0  +MOVJ EC00102
SREFP 3 C00103 BC00103  +REFP EC00103
CALL JOB:SEARCH-R1-S13D
SET P044 P006
SFTON3D P044
SMOVL C00104 BC00104 V=100.0  +MOVJ EC00104
SFTOF3D
MOVJ C00105 BC00105 VJ=100.00  +MOVJ EC00105 VJ=100.00
MOVJ C00106 BC00106 VJ=100.00  +MOVJ EC00106 VJ=100.00
MOVJ C00107 BC00107 VJ=100.00  +MOVJ EC00107 VJ=100.00
MOVJ C00108 BC00108 VJ=100.00  +MOVJ EC00108 VJ=100.00
SMOVL C00109 BC00109 V=100.0  +MOVJ EC00109
SREFP 3 C00110 BC00110  +REFP EC00110
CALL JOB:SEARCH-R1-S13D
SET P037 P006
SFTON3D P037
SMOVL C00111 BC00111 V=100.0  +MOVJ EC00111
SREFP 3 C00112 BC00112  +REFP EC00112
CALL JOB:SEARCH-R1-S13D
SET P037 P006
SFTON3D P037
SMOVL C00113 BC00113 V=100.0  +MOVJ EC00113
SFTOF3D
MOVJ C00114 BC00114 VJ=100.00  +MOVJ EC00114 VJ=100.00
SMOVL C00115 BC00115 V=100.0  +MOVJ EC00115
SREFP 3 C00116 BC00116  +REFP EC00116
CALL JOB:SEARCH-R1-S13D
SET P038 P006
SFTON3D P038
SMOVL C00117 BC00117 V=100.0  +MOVJ EC00117
SREFP 3 C00118 BC00118  +REFP EC00118
CALL JOB:SEARCH-R1-S13D
SET P038 P006
SFTON3D P038
SMOVL C00119 BC00119 V=100.0  +MOVJ EC00119
SFTOF3D
MOVJ C00120 BC00120 VJ=100.00  +MOVJ EC00120 VJ=100.00
MOVJ C00121 BC00121 VJ=100.00  +MOVJ EC00121 VJ=100.00
MOVJ C00122 BC00122 VJ=100.00  +MOVJ EC00122 VJ=100.00
MOVJ C00123 BC00123 VJ=100.00  +MOVJ EC00123 VJ=100.00
SMOVL C00124 BC00124 V=100.0  +MOVJ EC00124
SREFP 3 C00125 BC00125  +REFP EC00125
CALL JOB:SEARCH-R1-S13D
SET P039 P006
SFTON3D P039
SMOVL C00126 BC00126 V=100.0  +MOVJ EC00126
SREFP 3 C00127 BC00127  +REFP EC00127
CALL JOB:SEARCH-R1-S13D
SET P039 P006
SFTON3D P039
SMOVL C00128 BC00128 V=100.0  +MOVJ EC00128
SFTOF3D
MOVJ C00129 BC00129 VJ=100.00  +MOVJ EC00129 VJ=100.00
SMOVL C00130 BC00130 V=100.0  +MOVJ EC00130
SREFP 3 C00131 BC00131  +REFP EC00131
CALL JOB:SEARCH-R1-S13D
SET P040 P006
SFTON3D P040
SMOVL C00132 BC00132 V=100.0  +MOVJ EC00132
SREFP 3 C00133 BC00133  +REFP EC00133
CALL JOB:SEARCH-R1-S13D
SET P040 P006
SFTON3D P040
SMOVL C00134 BC00134 V=100.0  +MOVJ EC00134
MOVJ C00135 BC00135 VJ=100.00  +MOVJ EC00135 VJ=100.00
SFTOF3D
MOVJ C00136 BC00136 VJ=100.00  +MOVJ EC00136 VJ=100.00
MOVJ C00137 BC00137 VJ=100.00  +MOVJ EC00137 VJ=100.00
SMOVL C00138 BC00138 V=100.0  +MOVJ EC00138
SREFP 3 C00139 BC00139  +REFP EC00139
CALL JOB:SEARCH-R1-S13D
SET P041 P006
SFTON3D P041
SMOVL C00140 BC00140 V=100.0  +MOVJ EC00140
SREFP 3 C00141 BC00141  +REFP EC00141
CALL JOB:SEARCH-R1-S13D
SET P041 P006
SFTON3D P041
SMOVL C00142 BC00142 V=100.0  +MOVJ EC00142
SFTOF3D
MOVJ C00143 BC00143 VJ=100.00  +MOVJ EC00143 VJ=100.00
SMOVL C00144 BC00144 V=100.0  +MOVJ EC00144
SREFP 3 C00145 BC00145  +REFP EC00145
CALL JOB:SEARCH-R1-S13D
SET P042 P006
SFTON3D P042
SMOVL C00146 BC00146 V=100.0  +MOVJ EC00146
SREFP 3 C00147 BC00147  +REFP EC00147
CALL JOB:SEARCH-R1-S13D
SET P042 P006
SFTON3D P042
SMOVL C00148 BC00148 V=250.0  +MOVJ EC00148
MOVJ C00149 BC00149 VJ=100.00  +MOVJ EC00149 VJ=100.00
SFTOF3D
MOVJ C00150 BC00150 VJ=100.00  +MOVJ EC00150 VJ=100.00
SMOVL C00151 BC00151 V=100.0  +MOVJ EC00151
SREFP 3 C00152 BC00152  +REFP EC00152
CALL JOB:SEARCH-R1-S13D
SET P043 P006
SFTON3D P043
SMOVL C00153 BC00153 V=100.0  +MOVJ EC00153
SREFP 3 C00154 BC00154  +REFP EC00154
CALL JOB:SEARCH-R1-S13D
SET P043 P006
SFTON3D P043
SMOVL C00155 BC00155 V=166.7  +MOVJ EC00155
'KONIEC POMIARU
SMOVL C00156 BC00156 V=166.7  +MOVJ EC00156
MACRO1 MJ#(0) ARGF9
SFTON3D P043
SMOVL C00157 BC00157 V=250.0  +MOVJ EC00157
ARCON
SWVON WEV#(30)
SMOVL C00158 BC00158 V=10.0  +MOVJ EC00158
SMOVL C00159 BC00159 V=10.0  +MOVJ EC00159
SMOVL C00160 BC00160 V=10.0  +MOVJ EC00160
ARCOF
SWVOF
SFTOF3D
MOVJ C00161 BC00161 VJ=15.00  +MOVJ EC00161 VJ=100.00
MOVJ C00162 BC00162 VJ=100.00  +MOVJ EC00162 VJ=100.00
MOVJ C00163 BC00163 VJ=100.00  +MOVJ EC00163 VJ=100.00
MOVJ C00164 BC00164 VJ=100.00  +MOVJ EC00164 VJ=100.00
SFTON3D P044
SMOVL C00165 BC00165 V=166.7 PL=0  +MOVJ EC00165
ARCON
SWVON WEV#(30)
SMOVL C00166 BC00166 V=8.3  +MOVJ EC00166
SMOVL C00167 BC00167 V=8.3  +MOVJ EC00167
SMOVL C00168 BC00168 V=8.3  +MOVJ EC00168
ARCOF
SWVOF
SFTOF3D
MOVJ C00169 BC00169 VJ=15.00  +MOVJ EC00169 VJ=15.00
MOVJ C00170 BC00170 VJ=100.00  +MOVJ EC00170 VJ=100.00
MACRO1 MJ#(0) ARGF9
SFTON3D P031
SMOVL C00171 BC00171 V=133.3  +MOVJ EC00171
ARCON
SWVON WEV#(10)
SMOVL C00172 BC00172 V=10.0  +MOVJ EC00172
SFTON3D P030
SMOVL C00173 BC00173 V=10.0  +MOVJ EC00173
SMOVL C00174 BC00174 V=10.0  +MOVJ EC00174
ARCOF
SWVOF
SFTOF
MOVJ C00175 BC00175 VJ=100.00  +MOVJ EC00175 VJ=100.00
MOVJ C00176 BC00176 VJ=100.00  +MOVJ EC00176 VJ=100.00
MOVJ C00177 BC00177 VJ=100.00  +MOVJ EC00177 VJ=100.00
SFTON3D P038
SMOVL C00178 BC00178 V=166.7  +MOVJ EC00178
ARCON
SFTON3D P037
MOVL C00179 BC00179 V=9.2  +MOVJ EC00179 VJ=100.00
ARCOF
TIMER T=1.00
SFTOF3D
MOVJ C00180 BC00180 VJ=100.00  +MOVJ EC00180 VJ=100.00
MOVJ C00181 BC00181 VJ=100.00  +MOVJ EC00181 VJ=100.00
MOVJ C00182 BC00182 VJ=100.00  +MOVJ EC00182 VJ=100.00
MOVJ C00183 BC00183 VJ=100.00  +MOVJ EC00183 VJ=100.00
MACRO1 MJ#(0) ARGF14
MOVJ C00184 BC00184 VJ=100.00  +MOVJ EC00184 VJ=100.00
SFTON3D P041
SMOVL C00185 BC00185 V=166.7  +MOVJ EC00185
ARCON
SMOVL C00186 BC00186 V=9.2  +MOVJ EC00186
SFTON3D P042
SMOVL C00187 BC00187 V=9.2  +MOVJ EC00187
ARCOF
SFTOF3D
MOVJ C00188 BC00188 VJ=100.00  +MOVJ EC00188 VJ=100.00
MOVJ C00189 BC00189 VJ=100.00  +MOVJ EC00189 VJ=100.00
SFTON3D P040
SMOVL C00190 BC00190 V=166.7  +MOVJ EC00190
ARCON
SMOVL C00191 BC00191 V=9.2  +MOVJ EC00191
SFTON3D P039
SMOVL C00192 BC00192 V=9.2  +MOVJ EC00192
SMOVL C00193 BC00193 V=9.2  +MOVJ EC00193
ARCOF
SFTOF3D
MOVJ C00194 BC00194 VJ=100.00  +MOVJ EC00194 VJ=100.00
MOVJ C00195 BC00195 VJ=100.00  +MOVJ EC00195 VJ=100.00
MOVJ C00196 BC00196 VJ=100.00  +MOVJ EC00196 VJ=100.00
MOVJ C00197 BC00197 VJ=100.00  +MOVJ EC00197 VJ=100.00
MACRO1 MJ#(0) ARGF9
SFTON3D P036
SMOVL C00198 BC00198 V=166.7  +MOVJ EC00198
ARCON
SMOVL C00199 BC00199 V=9.2  +MOVJ EC00199
SFTON3D P035
SMOVL C00200 BC00200 V=9.2  +MOVJ EC00200
SMOVL C00201 BC00201 V=9.2  +MOVJ EC00201
ARCOF
SFTOF3D
MOVJ C00202 BC00202 VJ=15.00  +MOVJ EC00202 VJ=100.00
MOVJ C00203 BC00203 VJ=100.00  +MOVJ EC00203 VJ=15.00
MACRO1 MJ#(0) ARGF9
SFTON3D P034
SMOVL C00204 BC00204 V=166.7  +MOVJ EC00204
ARCON
SMOVC C00205 BC00205 V=8.3  +MOVJ EC00205
SMOVC C00206 BC00206 V=8.3  +MOVJ EC00206
SMOVC C00207 BC00207 V=8.3  +MOVJ EC00207
SMOVL C00208 BC00208 V=10.0  +MOVJ EC00208
SMOVC C00209 BC00209 V=8.3  +MOVJ EC00209
SMOVC C00210 BC00210 V=8.3  +MOVJ EC00210
SMOVC C00211 BC00211 V=8.3  +MOVJ EC00211
ARCOF
SFTOF3D
MOVJ C00212 BC00212 VJ=100.00  +MOVJ EC00212 VJ=100.00
MOVJ C00213 BC00213 VJ=100.00  +MOVJ EC00213 VJ=100.00
SFTON3D P032
SMOVL C00214 BC00214 V=250.0  +MOVJ EC00214
ARCON
SMOVL C00215 BC00215 V=8.3  +MOVJ EC00215
SFTON3D P033
SMOVL C00216 BC00216 V=8.3  +MOVJ EC00216
SMOVL C00217 BC00217 V=8.3  +MOVJ EC00217
ARCOF
SFTOF3D
MOVJ C00218 BC00218 VJ=30.00  +MOVJ EC00218 VJ=100.00
MOVJ C00219 BC00219 VJ=30.00  +MOVJ EC00219 VJ=15.00
JUMP *LABEL
'Up
'Path S1856
SFTOF3D
MOVJ C00220 BC00220 VJ=100.00  +MOVJ EC00220 VJ=100.00
COMM MOVL C00221 BC00221 V=400.0  +MOVJ EC00221 VJ=100.00
COMM SMOVL C00222 BC00222 V=60.0  +MOVJ EC00222
COMM SREFP 3 C00223 BC00223  +REFP EC00223
COMM CALL JOB:SEARCH-R1-S13D
COMM SET P042 P006
COMM SFTON3D P042
COMM SMOVL C00224 BC00224 V=60.0  +MOVJ EC00224
COMM SMOVL C00225 BC00225 V=60.0  +MOVJ EC00225
COMM SREFP 3 C00226 BC00226  +REFP EC00226
COMM CALL JOB:SEARCH-R1-S13D
COMM SET P042 P006
COMM SFTON3D P042
COMM SMOVL C00227 BC00227 V=60.0  +MOVJ EC00227
COMM MOVL C00228 BC00228 V=400.0  +MOVJ EC00228 VJ=100.00
COMM MOVL C00229 BC00229 V=1000.0  +MOVJ EC00229 VJ=100.00
COMM 'Path S1857
COMM SFTOF3D
COMM MOVJ C00230 BC00230 VJ=100.00  +MOVJ EC00230 VJ=100.00
COMM MOVL C00231 BC00231 V=400.0  +MOVJ EC00231 VJ=100.00
COMM SMOVL C00232 BC00232 V=60.0  +MOVJ EC00232
COMM SREFP 3 C00233 BC00233  +REFP EC00233
COMM CALL JOB:SEARCH-R1-S13D
COMM SET P041 P006
COMM SFTON3D P041
COMM SMOVL C00234 BC00234 V=60.0  +MOVJ EC00234
COMM SMOVL C00235 BC00235 V=60.0  +MOVJ EC00235
COMM SREFP 3 C00236 BC00236  +REFP EC00236
COMM CALL JOB:SEARCH-R1-S13D
COMM SET P041 P006
COMM SFTON3D P041
COMM SMOVL C00237 BC00237 V=60.0  +MOVJ EC00237
COMM MOVL C00238 BC00238 V=400.0  +MOVJ EC00238 VJ=100.00
COMM MOVL C00239 BC00239 V=1000.0  +MOVJ EC00239 VJ=100.00
COMM 'Path S1858
COMM SFTOF3D
COMM MOVJ C00240 BC00240 VJ=100.00  +MOVJ EC00240 VJ=100.00
COMM MOVL C00241 BC00241 V=400.0  +MOVJ EC00241 VJ=100.00
COMM SMOVL C00242 BC00242 V=60.0  +MOVJ EC00242
COMM SREFP 3 C00243 BC00243  +REFP EC00243
COMM CALL JOB:SEARCH-R1-S13D
COMM SET P040 P006
COMM SFTON3D P040
COMM SMOVL C00244 BC00244 V=60.0  +MOVJ EC00244
COMM SMOVL C00245 BC00245 V=60.0  +MOVJ EC00245
COMM SREFP 3 C00246 BC00246  +REFP EC00246
COMM CALL JOB:SEARCH-R1-S13D
COMM SET P040 P006
COMM SFTON3D P040
COMM SMOVL C00247 BC00247 V=60.0  +MOVJ EC00247
COMM MOVL C00248 BC00248 V=400.0  +MOVJ EC00248 VJ=100.00
COMM MOVL C00249 BC00249 V=1000.0  +MOVJ EC00249 VJ=100.00
MOVL C00250 BC00250 V=1000.0  +MOVJ EC00250 VJ=100.00
'Path S1859
SFTOF3D
MOVJ C00251 BC00251 VJ=100.00  +MOVJ EC00251 VJ=100.00
MOVJ C00252 BC00252 VJ=100.00  +MOVJ EC00252 VJ=100.00
MOVL C00253 BC00253 V=400.0  +MOVJ EC00253 VJ=100.00
SMOVL C00254 BC00254 V=60.0  +MOVJ EC00254
SREFP 3 C00255 BC00255  +REFP EC00255
CALL JOB:SEARCH-R1-S13D
SET P043 P006
SFTON3D P043
SMOVL C00256 BC00256 V=60.0  +MOVJ EC00256
SMOVL C00257 BC00257 V=60.0  +MOVJ EC00257
SREFP 3 C00258 BC00258  +REFP EC00258
CALL JOB:SEARCH-R1-S13D
SET P043 P006
SFTON3D P043
SMOVL C00259 BC00259 V=60.0  +MOVJ EC00259
MOVL C00260 BC00260 V=400.0  +MOVJ EC00260 VJ=100.00
MOVL C00261 BC00261 V=1000.0  +MOVJ EC00261 VJ=100.00
'Path S1860
SFTOF3D
MOVJ C00262 BC00262 VJ=100.00  +MOVJ EC00262 VJ=100.00
MOVL C00263 BC00263 V=400.0  +MOVJ EC00263 VJ=100.00
SMOVL C00264 BC00264 V=60.0  +MOVJ EC00264
SREFP 3 C00265 BC00265  +REFP EC00265
CALL JOB:SEARCH-R1-S13D
SET P039 P006
SFTON3D P039
SMOVL C00266 BC00266 V=60.0  +MOVJ EC00266
SMOVL C00267 BC00267 V=60.0  +MOVJ EC00267
SREFP 3 C00268 BC00268  +REFP EC00268
CALL JOB:SEARCH-R1-S13D
SET P039 P006
SFTON3D P039
SMOVL C00269 BC00269 V=60.0  +MOVJ EC00269
MOVL C00270 BC00270 V=400.0  +MOVJ EC00270 VJ=100.00
MOVL C00271 BC00271 V=1000.0  +MOVJ EC00271 VJ=100.00
MOVJ C00272 BC00272 VJ=100.00  +MOVJ EC00272 VJ=100.00
'Path S1861
SFTOF3D
MOVJ C00273 BC00273 VJ=100.00  +MOVJ EC00273 VJ=100.00
MOVL C00274 BC00274 V=400.0  +MOVJ EC00274 VJ=100.00
SMOVL C00275 BC00275 V=60.0  +MOVJ EC00275
SREFP 3 C00276 BC00276  +REFP EC00276
CALL JOB:SEARCH-R1-S13D
SET P034 P006
SFTON3D P034
SMOVL C00277 BC00277 V=60.0  +MOVJ EC00277
SMOVL C00278 BC00278 V=60.0  +MOVJ EC00278
SREFP 3 C00279 BC00279  +REFP EC00279
CALL JOB:SEARCH-R1-S13D
SET P034 P006
SFTON3D P034
SMOVL C00280 BC00280 V=60.0  +MOVJ EC00280
MOVL C00281 BC00281 V=400.0  +MOVJ EC00281 VJ=100.00
MOVL C00282 BC00282 V=1000.0  +MOVJ EC00282 VJ=100.00
MOVJ C00283 BC00283 VJ=100.00  +MOVJ EC00283 VJ=100.00
'Path S1862
SFTOF3D
MOVJ C00284 BC00284 VJ=100.00  +MOVJ EC00284 VJ=100.00
MOVL C00285 BC00285 V=400.0  +MOVJ EC00285 VJ=100.00
SMOVL C00286 BC00286 V=60.0  +MOVJ EC00286
SREFP 3 C00287 BC00287  +REFP EC00287
CALL JOB:SEARCH-R1-S13D
SET P038 P006
SFTON3D P038
SMOVL C00288 BC00288 V=60.0  +MOVJ EC00288
SMOVL C00289 BC00289 V=60.0  +MOVJ EC00289
SREFP 3 C00290 BC00290  +REFP EC00290
CALL JOB:SEARCH-R1-S13D
SET P038 P006
SFTON3D P038
SMOVL C00291 BC00291 V=60.0  +MOVJ EC00291
SMOVL C00292 BC00292 V=60.0  +MOVJ EC00292
SREFP 3 C00293 BC00293  +REFP EC00293
CALL JOB:SEARCH-R1-S13D
SET P038 P006
SFTON3D P038
SMOVL C00294 BC00294 V=60.0  +MOVJ EC00294
MOVL C00295 BC00295 V=400.0  +MOVJ EC00295 VJ=100.00
MOVL C00296 BC00296 V=1000.0  +MOVJ EC00296 VJ=100.00
'Path S1863
SFTOF3D
MOVJ C00297 BC00297 VJ=100.00  +MOVJ EC00297 VJ=100.00
MOVL C00298 BC00298 V=400.0  +MOVJ EC00298 VJ=100.00
SMOVL C00299 BC00299 V=60.0  +MOVJ EC00299
SREFP 3 C00300 BC00300  +REFP EC00300
CALL JOB:SEARCH-R1-S13D
SET P033 P006
SFTON3D P033
SMOVL C00301 BC00301 V=60.0  +MOVJ EC00301
SMOVL C00302 BC00302 V=60.0  +MOVJ EC00302
SREFP 3 C00303 BC00303  +REFP EC00303
CALL JOB:SEARCH-R1-S13D
SET P033 P006
SFTON3D P033
SMOVL C00304 BC00304 V=60.0  +MOVJ EC00304
MOVL C00305 BC00305 V=400.0  +MOVJ EC00305 VJ=100.00
MOVL C00306 BC00306 V=1000.0  +MOVJ EC00306 VJ=100.00
MOVL C00307 BC00307 V=1000.0  +MOVJ EC00307 VJ=100.00
'Path S1864
SFTOF3D
MOVJ C00308 BC00308 VJ=100.00  +MOVJ EC00308 VJ=100.00
MOVJ C00309 BC00309 VJ=100.00  +MOVJ EC00309 VJ=100.00
MOVL C00310 BC00310 V=400.0  +MOVJ EC00310 VJ=100.00
SMOVL C00311 BC00311 V=60.0  +MOVJ EC00311
SREFP 3 C00312 BC00312  +REFP EC00312
CALL JOB:SEARCH-R1-S13D
SET P035 P006
SFTON3D P035
SMOVL C00313 BC00313 V=60.0  +MOVJ EC00313
SMOVL C00314 BC00314 V=60.0  +MOVJ EC00314
SREFP 3 C00315 BC00315  +REFP EC00315
CALL JOB:SEARCH-R1-S13D
SET P035 P006
SFTON3D P035
SMOVL C00316 BC00316 V=60.0  +MOVJ EC00316
MOVL C00317 BC00317 V=400.0  +MOVJ EC00317 VJ=100.00
MOVL C00318 BC00318 V=1000.0  +MOVJ EC00318 VJ=100.00
MOVL C00319 BC00319 V=1000.0  +MOVJ EC00319 VJ=100.00
'Path S1865
SFTOF3D
MOVJ C00320 BC00320 VJ=100.00  +MOVJ EC00320 VJ=100.00
MOVL C00321 BC00321 V=400.0  +MOVJ EC00321 VJ=100.00
SMOVL C00322 BC00322 V=60.0  +MOVJ EC00322
SREFP 3 C00323 BC00323  +REFP EC00323
CALL JOB:SEARCH-R1-S13D
SET P037 P006
SFTON3D P037
SMOVL C00324 BC00324 V=60.0  +MOVJ EC00324
SMOVL C00325 BC00325 V=60.0  +MOVJ EC00325
SREFP 3 C00326 BC00326  +REFP EC00326
CALL JOB:SEARCH-R1-S13D
SET P037 P006
SFTON3D P037
SMOVL C00327 BC00327 V=60.0  +MOVJ EC00327
MOVL C00328 BC00328 V=400.0  +MOVJ EC00328 VJ=100.00
MOVL C00329 BC00329 V=1000.0  +MOVJ EC00329 VJ=100.00
'Path S1866
SFTOF3D
MOVJ C00330 BC00330 VJ=100.00  +MOVJ EC00330 VJ=100.00
MOVJ C00331 BC00331 VJ=100.00  +MOVJ EC00331 VJ=100.00
MOVL C00332 BC00332 V=400.0  +MOVJ EC00332 VJ=100.00
SMOVL C00333 BC00333 V=60.0  +MOVJ EC00333
SREFP 3 C00334 BC00334  +REFP EC00334
CALL JOB:SEARCH-R1-S13D
SET P031 P006
SFTON3D P031
SMOVL C00335 BC00335 V=60.0  +MOVJ EC00335
SMOVL C00336 BC00336 V=60.0  +MOVJ EC00336
SREFP 3 C00337 BC00337  +REFP EC00337
CALL JOB:SEARCH-R1-S13D
SET P031 P006
SFTON3D P031
SMOVL C00338 BC00338 V=60.0  +MOVJ EC00338
MOVL C00339 BC00339 V=400.0  +MOVJ EC00339 VJ=100.00
MOVL C00340 BC00340 V=1000.0  +MOVJ EC00340 VJ=100.00
'Path S1867
MOVJ C00341 BC00341 VJ=20.00  +MOVJ EC00341 VJ=20.00
MOVJ C00342 BC00342 VJ=20.00  +MOVJ EC00342 VJ=20.00
SFTOF3D
MOVJ C00343 BC00343 VJ=100.00  +MOVJ EC00343 VJ=100.00
MOVL C00344 BC00344 V=400.0  +MOVJ EC00344 VJ=100.00
SMOVL C00345 BC00345 V=60.0  +MOVJ EC00345
SREFP 3 C00346 BC00346  +REFP EC00346
CALL JOB:SEARCH-R1-S13D
SET P036 P006
SFTON3D P036
SMOVL C00347 BC00347 V=60.0  +MOVJ EC00347
SMOVL C00348 BC00348 V=60.0  +MOVJ EC00348
SREFP 3 C00349 BC00349  +REFP EC00349
CALL JOB:SEARCH-R1-S13D
SET P036 P006
SFTON3D P036
SMOVL C00350 BC00350 V=60.0  +MOVJ EC00350
MOVL C00351 BC00351 V=400.0  +MOVJ EC00351 VJ=100.00
MOVL C00352 BC00352 V=1000.0  +MOVJ EC00352 VJ=100.00
MOVL C00353 BC00353 V=1000.0  +MOVJ EC00353 VJ=100.00
'Path S1868
SFTOF3D
MOVJ C00354 BC00354 VJ=100.00  +MOVJ EC00354 VJ=100.00
MOVL C00355 BC00355 V=400.0  +MOVJ EC00355 VJ=100.00
SMOVL C00356 BC00356 V=60.0  +MOVJ EC00356
SREFP 3 C00357 BC00357  +REFP EC00357
CALL JOB:SEARCH-R1-S13D
SET P032 P006
SFTON3D P032
SMOVL C00358 BC00358 V=60.0  +MOVJ EC00358
SMOVL C00359 BC00359 V=60.0  +MOVJ EC00359
SREFP 3 C00360 BC00360  +REFP EC00360
CALL JOB:SEARCH-R1-S13D
SET P032 P006
SFTON3D P032
SMOVL C00361 BC00361 V=60.0  +MOVJ EC00361
MOVL C00362 BC00362 V=400.0  +MOVJ EC00362 VJ=100.00
MOVL C00363 BC00363 V=1000.0  +MOVJ EC00363 VJ=100.00
'Path W1869
SFTOF3D
SFTON3D P032
MOVJ C00364 BC00364 VJ=100.00  +MOVJ EC00364 VJ=100.00
SMOVL C00365 BC00365 V=400.0  +MOVJ EC00365
SMOVL C00366 BC00366 V=100.0 PL=0  +MOVJ EC00366
SREFP 1 C00367 BC00367  +REFP EC00367
SREFP 2 C00368 BC00368  +REFP EC00368
MACRO1 MJ#(0) ARGF0
ARCON
SMOVL C00369 BC00369 V=10.0  +MOVJ EC00369
SMOVL C00370 BC00370 V=10.0  +MOVJ EC00370
SMOVL C00371 BC00371 V=10.0  +MOVJ EC00371
ARCOF
SMOVL C00372 BC00372 V=400.0  +MOVJ EC00372
SMOVL C00373 BC00373 V=1000.0  +MOVJ EC00373
SMOVL C00374 BC00374 V=1000.0  +MOVJ EC00374
SFTOF3D
MOVJ C00375 BC00375 VJ=100.00  +MOVJ EC00375 VJ=100.00
'Path W1870
SFTOF3D
SFTON3D P033
MOVJ C00376 BC00376 VJ=100.00  +MOVJ EC00376 VJ=100.00
MOVJ C00377 BC00377 VJ=100.00  +MOVJ EC00377 VJ=100.00
SMOVL C00378 BC00378 V=400.0  +MOVJ EC00378
SMOVL C00379 BC00379 V=100.0 PL=0  +MOVJ EC00379
SREFP 1 C00380 BC00380  +REFP EC00380
SREFP 2 C00381 BC00381  +REFP EC00381
MACRO1 MJ#(0) ARGF0
ARCON
SMOVL C00382 BC00382 V=10.0  +MOVJ EC00382
SMOVL C00383 BC00383 V=10.0  +MOVJ EC00383
SMOVL C00384 BC00384 V=10.0  +MOVJ EC00384
ARCOF
SMOVL C00385 BC00385 V=400.0  +MOVJ EC00385
SMOVL C00386 BC00386 V=1000.0  +MOVJ EC00386
SFTOF3D
'Path W1871
SFTOF3D
SFTON3D P034
MOVJ C00387 BC00387 VJ=100.00  +MOVJ EC00387 VJ=100.00
SMOVL C00388 BC00388 V=400.0  +MOVJ EC00388
SMOVL C00389 BC00389 V=100.0 PL=0  +MOVJ EC00389
SREFP 1 C00390 BC00390  +REFP EC00390
SREFP 2 C00391 BC00391  +REFP EC00391
MACRO1 MJ#(0) ARGF0
ARCON
SMOVL C00392 BC00392 V=10.0  +MOVJ EC00392
SMOVL C00393 BC00393 V=10.0  +MOVJ EC00393
ARCOF
SMOVL C00394 BC00394 V=400.0  +MOVJ EC00394
SMOVL C00395 BC00395 V=1000.0  +MOVJ EC00395
SMOVL C00396 BC00396 V=1000.0  +MOVJ EC00396
SFTOF3D
MOVJ C00397 BC00397 VJ=20.00  +MOVJ EC00397 VJ=20.00
MOVJ C00398 BC00398 VJ=20.00  +MOVJ EC00398 VJ=20.00
'Path W1872
SFTOF3D
SFTON3D P031
MOVJ C00399 BC00399 VJ=100.00  +MOVJ EC00399 VJ=100.00
SMOVL C00400 BC00400 V=400.0  +MOVJ EC00400
SMOVL C00401 BC00401 V=100.0 PL=0  +MOVJ EC00401
SREFP 1 C00402 BC00402  +REFP EC00402
SREFP 2 C00403 BC00403  +REFP EC00403
MACRO1 MJ#(0) ARGF0
ARCON
SMOVL C00404 BC00404 V=10.0  +MOVJ EC00404
SMOVL C00405 BC00405 V=10.0  +MOVJ EC00405
ARCOF
SMOVL C00406 BC00406 V=400.0  +MOVJ EC00406
SMOVL C00407 BC00407 V=1000.0  +MOVJ EC00407
SMOVL C00408 BC00408 V=1000.0  +MOVJ EC00408
SFTOF3D
'Path W1873
MOVJ C00409 BC00409 VJ=20.00  +MOVJ EC00409 VJ=20.00
SFTOF3D
SFTON3D P035
MOVJ C00410 BC00410 VJ=100.00  +MOVJ EC00410 VJ=100.00
SMOVL C00411 BC00411 V=400.0  +MOVJ EC00411
SMOVL C00412 BC00412 V=100.0 PL=0  +MOVJ EC00412
SREFP 1 C00413 BC00413  +REFP EC00413
SREFP 2 C00414 BC00414  +REFP EC00414
MACRO1 MJ#(0) ARGF0
ARCON
SMOVL C00415 BC00415 V=10.0  +MOVJ EC00415
SMOVL C00416 BC00416 V=10.0  +MOVJ EC00416
ARCOF
SMOVL C00417 BC00417 V=400.0  +MOVJ EC00417
SMOVL C00418 BC00418 V=1000.0  +MOVJ EC00418
SMOVL C00419 BC00419 V=1000.0  +MOVJ EC00419
SFTOF3D
MOVJ C00420 BC00420 VJ=100.00  +MOVJ EC00420 VJ=100.00
'Path W1874
SFTOF3D
SFTON3D P036
MOVJ C00421 BC00421 VJ=100.00  +MOVJ EC00421 VJ=100.00
SMOVL C00422 BC00422 V=400.0  +MOVJ EC00422
SMOVL C00423 BC00423 V=100.0 PL=0  +MOVJ EC00423
SREFP 1 C00424 BC00424  +REFP EC00424
SREFP 2 C00425 BC00425  +REFP EC00425
MACRO1 MJ#(0) ARGF0
ARCON
SMOVL C00426 BC00426 V=10.0  +MOVJ EC00426
SMOVL C00427 BC00427 V=10.0  +MOVJ EC00427
SMOVL C00428 BC00428 V=10.0  +MOVJ EC00428
ARCOF
SMOVL C00429 BC00429 V=400.0  +MOVJ EC00429
SMOVL C00430 BC00430 V=1000.0  +MOVJ EC00430
SMOVL C00431 BC00431 V=1000.0  +MOVJ EC00431
SFTOF3D
MOVJ C00432 BC00432 VJ=100.00  +MOVJ EC00432 VJ=100.00
'Path W1875
SFTOF3D
SFTON3D P037
MOVJ C00433 BC00433 VJ=100.00  +MOVJ EC00433 VJ=100.00
MOVJ C00434 BC00434 VJ=100.00  +MOVJ EC00434 VJ=100.00
SMOVL C00435 BC00435 V=400.0  +MOVJ EC00435
SMOVL C00436 BC00436 V=100.0 PL=0  +MOVJ EC00436
SREFP 1 C00437 BC00437  +REFP EC00437
SREFP 2 C00438 BC00438  +REFP EC00438
MACRO1 MJ#(0) ARGF0
ARCON
SMOVL C00439 BC00439 V=10.0  +MOVJ EC00439
SMOVL C00440 BC00440 V=10.0  +MOVJ EC00440
SMOVL C00441 BC00441 V=10.0  +MOVJ EC00441
ARCOF
SMOVL C00442 BC00442 V=400.0  +MOVJ EC00442
SMOVL C00443 BC00443 V=1000.0  +MOVJ EC00443
SMOVL C00444 BC00444 V=1000.0  +MOVJ EC00444
SFTOF3D
MOVJ C00445 BC00445 VJ=100.00  +MOVJ EC00445 VJ=100.00
'Path W1876
SFTOF3D
SFTON3D P038
MOVJ C00446 BC00446 VJ=100.00  +MOVJ EC00446 VJ=100.00
MOVJ C00447 BC00447 VJ=100.00  +MOVJ EC00447 VJ=100.00
SMOVL C00448 BC00448 V=400.0  +MOVJ EC00448
SMOVL C00449 BC00449 V=100.0 PL=0  +MOVJ EC00449
SREFP 1 C00450 BC00450  +REFP EC00450
SREFP 2 C00451 BC00451  +REFP EC00451
MACRO1 MJ#(0) ARGF0
ARCON
SMOVL C00452 BC00452 V=10.0  +MOVJ EC00452
SMOVL C00453 BC00453 V=10.0  +MOVJ EC00453
ARCOF
SMOVL C00454 BC00454 V=400.0  +MOVJ EC00454
SMOVL C00455 BC00455 V=1000.0  +MOVJ EC00455
SFTOF3D
'Path W1877
SFTOF3D
SFTON3D P038
SMOVL C00456 BC00456 V=400.0  +MOVJ EC00456
SMOVL C00457 BC00457 V=100.0 PL=0  +MOVJ EC00457
SREFP 1 C00458 BC00458  +REFP EC00458
SREFP 2 C00459 BC00459  +REFP EC00459
MACRO1 MJ#(0) ARGF0
ARCON
SMOVL C00460 BC00460 V=10.0  +MOVJ EC00460
SMOVL C00461 BC00461 V=10.0  +MOVJ EC00461
SMOVL C00462 BC00462 V=10.0  +MOVJ EC00462
ARCOF
SMOVL C00463 BC00463 V=400.0  +MOVJ EC00463
SFTOF3D
MOVJ C00464 BC00464 VJ=100.00  +MOVJ EC00464 VJ=100.00
'Path W1878
SFTOF3D
SFTON3D P039
MOVJ C00465 BC00465 VJ=100.00  +MOVJ EC00465 VJ=100.00
MOVJ C00466 BC00466 VJ=100.00  +MOVJ EC00466 VJ=100.00
SMOVL C00467 BC00467 V=400.0  +MOVJ EC00467
SMOVL C00468 BC00468 V=100.0 PL=0  +MOVJ EC00468
SREFP 1 C00469 BC00469  +REFP EC00469
SREFP 2 C00470 BC00470  +REFP EC00470
MACRO1 MJ#(0) ARGF0
ARCON
SMOVL C00471 BC00471 V=10.0  +MOVJ EC00471
ARCOF
SMOVL C00472 BC00472 V=400.0  +MOVJ EC00472
SMOVL C00473 BC00473 V=1000.0  +MOVJ EC00473
SMOVL C00474 BC00474 V=1000.0  +MOVJ EC00474
SFTOF3D
'Path W1879
SFTOF3D
SFTON3D P042
MOVJ C00475 BC00475 VJ=100.00  +MOVJ EC00475 VJ=100.00
COMM MOVJ C00476 BC00476 VJ=100.00  +MOVJ EC00476 VJ=100.00
COMM SMOVL C00477 BC00477 V=400.0  +MOVJ EC00477
COMM SMOVL C00478 BC00478 V=100.0 PL=0  +MOVJ EC00478
COMM SREFP 1 C00479 BC00479  +REFP EC00479
COMM SREFP 2 C00480 BC00480  +REFP EC00480
COMM MACRO1 MJ#(0) ARGF0
COMM ARCON
COMM SMOVL C00481 BC00481 V=10.0  +MOVJ EC00481
COMM SMOVL C00482 BC00482 V=10.0  +MOVJ EC00482
COMM SMOVL C00483 BC00483 V=10.0  +MOVJ EC00483
COMM ARCOF
COMM SMOVL C00484 BC00484 V=400.0  +MOVJ EC00484
COMM SMOVL C00485 BC00485 V=1000.0  +MOVJ EC00485
SFTOF3D
'Path W1880
COMM SFTOF3D
COMM SFTON3D P041
COMM MOVJ C00486 BC00486 VJ=100.00  +MOVJ EC00486 VJ=100.00
COMM SMOVL C00487 BC00487 V=400.0  +MOVJ EC00487
COMM SMOVL C00488 BC00488 V=100.0 PL=0  +MOVJ EC00488
COMM SREFP 1 C00489 BC00489  +REFP EC00489
COMM SREFP 2 C00490 BC00490  +REFP EC00490
COMM MACRO1 MJ#(0) ARGF0
COMM ARCON
COMM SMOVL C00491 BC00491 V=10.0  +MOVJ EC00491
COMM ARCOF
COMM SMOVL C00492 BC00492 V=400.0  +MOVJ EC00492
COMM SMOVL C00493 BC00493 V=1000.0  +MOVJ EC00493
SFTOF3D
'Path W1881
COMM SFTOF3D
COMM SFTON3D P040
COMM MOVJ C00494 BC00494 VJ=100.00  +MOVJ EC00494 VJ=100.00
COMM SMOVL C00495 BC00495 V=400.0  +MOVJ EC00495
COMM SMOVL C00496 BC00496 V=100.0 PL=0  +MOVJ EC00496
COMM SREFP 1 C00497 BC00497  +REFP EC00497
COMM SREFP 2 C00498 BC00498  +REFP EC00498
COMM MACRO1 MJ#(0) ARGF0
COMM ARCON
COMM SMOVL C00499 BC00499 V=10.0  +MOVJ EC00499
COMM ARCOF
COMM SMOVL C00500 BC00500 V=400.0  +MOVJ EC00500
COMM SMOVL C00501 BC00501 V=1000.0  +MOVJ EC00501
COMM SMOVL C00502 BC00502 V=1000.0  +MOVJ EC00502
SFTOF3D
MOVJ C00503 BC00503 VJ=20.00  +MOVJ EC00503 VJ=20.00
'Path W1882
SFTOF3D
SFTON3D P043
MOVJ C00504 BC00504 VJ=100.00  +MOVJ EC00504 VJ=100.00
SMOVL C00505 BC00505 V=400.0  +MOVJ EC00505
SMOVL C00506 BC00506 V=100.0 PL=0  +MOVJ EC00506
SREFP 1 C00507 BC00507  +REFP EC00507
SREFP 2 C00508 BC00508  +REFP EC00508
MACRO1 MJ#(0) ARGF0
ARCON
COMM SMOVL C00509 BC00509 V=10.0  +MOVJ EC00509
COMM SMOVL C00510 BC00510 V=10.0  +MOVJ EC00510
COMM SMOVL C00511 BC00511 V=10.0  +MOVJ EC00511
COMM SMOVL C00512 BC00512 V=10.0  +MOVJ EC00512
COMM SMOVL C00513 BC00513 V=10.0  +MOVJ EC00513
COMM SMOVL C00514 BC00514 V=10.0  +MOVJ EC00514
COMM SMOVL C00515 BC00515 V=10.0  +MOVJ EC00515
SMOVL C00516 BC00516 V=10.0  +MOVJ EC00516
SMOVL C00517 BC00517 V=10.0  +MOVJ EC00517
SMOVL C00518 BC00518 V=10.0  +MOVJ EC00518
SMOVL C00519 BC00519 V=10.0  +MOVJ EC00519
SMOVL C00520 BC00520 V=10.0  +MOVJ EC00520
SMOVL C00521 BC00521 V=10.0  +MOVJ EC00521
SMOVL C00522 BC00522 V=10.0  +MOVJ EC00522
SMOVL C00523 BC00523 V=10.0  +MOVJ EC00523
ARCOF
SMOVL C00524 BC00524 V=400.0  +MOVJ EC00524
SMOVL C00525 BC00525 V=1000.0  +MOVJ EC00525
SFTOF3D
MOVJ C00526 BC00526 VJ=100.00  +MOVJ EC00526 VJ=100.00
MOVJ C00527 BC00527 VJ=100.00  +MOVJ EC00527 VJ=100.00
MOVJ C00528 BC00528 VJ=100.00  +MOVJ EC00528 VJ=100.00
*LABEL
'Down
MOVJ C00529 BC00529 VJ=50.00  +MOVJ EC00529 VJ=20.00
MOVJ C00530 BC00530 VJ=100.00  +MOVJ EC00530 VJ=100.00
MOVJ C00531 BC00531 VJ=100.00  +MOVJ EC00531 VJ=100.00
'1
'BRAKUJACY ELEMENT
'BRAKUJACY ELEMENT
'BRAKUJACY ELEMENT
'Path W1886
COMM SFTOF3D
COMM SFTON3D P023
COMM MOVJ C00532 BC00532 VJ=100.00  +MOVJ EC00532 VJ=100.00
COMM SMOVL C00533 BC00533 V=400.0  +MOVJ EC00533
COMM SMOVL C00534 BC00534 V=100.0 PL=0  +MOVJ EC00534
COMM SREFP 1 C00535 BC00535  +REFP EC00535
COMM SREFP 2 C00536 BC00536  +REFP EC00536
COMM MACRO1 MJ#(0) ARGF0
COMM ARCON
COMM SMOVL C00537 BC00537 V=10.0  +MOVJ EC00537
COMM SMOVL C00538 BC00538 V=10.0  +MOVJ EC00538
COMM SMOVL C00539 BC00539 V=10.0  +MOVJ EC00539
